BEGIN
   Zulauf_AR_Niv.Bef.BA_Nrm := FALSE;
   Zulauf_AR_Niv.Bef.BA_Frz := FALSE;
   Zulauf_AR_Niv.Bef.BA_EW := FALSE;
   Zulauf_AR_Niv.Bef.BA_Sim := FALSE;
   Zulauf_AR_Niv.Bef.BA_Wart := FALSE;
   Zulauf_AR_Niv.Bef.Frg_HH := FALSE;
   Zulauf_AR_Niv.Bef.Frg_H := FALSE;
   Zulauf_AR_Niv.Bef.Frg_L := FALSE;
   Zulauf_AR_Niv.Bef.Frg_LL := FALSE;
   Zulauf_AR_Niv.Bef.SB_MW_frz := FALSE;
   Zulauf_AR_Niv.Bef.SB_MW_EW := FALSE;
   Zulauf_AR_Niv.Bef.Res_11 := FALSE;
   Zulauf_AR_Niv.Bef.Res_12 := FALSE;
   Zulauf_AR_Niv.Bef.Res_13 := FALSE;
   Zulauf_AR_Niv.Bef.Res_14 := FALSE;
   Zulauf_AR_Niv.Bef.Res_15 := FALSE;
   Zulauf_AR_Niv.Bef.Res_16 := FALSE;
   Zulauf_AR_Niv.Bef.Res_17 := FALSE;
   Zulauf_AR_Niv.Bef.Res_18 := FALSE;
   Zulauf_AR_Niv.Bef.Res_19 := FALSE;
   Zulauf_AR_Niv.Bef.Res_20 := FALSE;
   Zulauf_AR_Niv.Bef.Res_21 := FALSE;
   Zulauf_AR_Niv.Bef.Res_22 := FALSE;
   Zulauf_AR_Niv.Bef.Res_23 := FALSE;
   Zulauf_AR_Niv.Bef.Res_24 := FALSE;
   Zulauf_AR_Niv.Bef.Res_25 := FALSE;
   Zulauf_AR_Niv.Bef.Res_26 := FALSE;
   Zulauf_AR_Niv.Bef.Res_27 := FALSE;
   Zulauf_AR_Niv.Bef.Res_28 := FALSE;
   Zulauf_AR_Niv.Bef.Res_29 := FALSE;
   Zulauf_AR_Niv.Bef.Res_30 := FALSE;
   Zulauf_AR_Niv.Bef.BF_Quit := FALSE;
   Zulauf_AR_Niv.MW_Sim := 8.0;
   Zulauf_AR_Temp.Bef.BA_Nrm := FALSE;
   Zulauf_AR_Temp.Bef.BA_Frz := FALSE;
   Zulauf_AR_Temp.Bef.BA_EW := FALSE;
   Zulauf_AR_Temp.Bef.BA_Sim := FALSE;
   Zulauf_AR_Temp.Bef.BA_Wart := FALSE;
   Zulauf_AR_Temp.Bef.Frg_HH := FALSE;
   Zulauf_AR_Temp.Bef.Frg_H := FALSE;
   Zulauf_AR_Temp.Bef.Frg_L := FALSE;
   Zulauf_AR_Temp.Bef.Frg_LL := FALSE;
   Zulauf_AR_Temp.Bef.SB_MW_frz := FALSE;
   Zulauf_AR_Temp.Bef.SB_MW_EW := FALSE;
   Zulauf_AR_Temp.Bef.Res_11 := FALSE;
   Zulauf_AR_Temp.Bef.Res_12 := FALSE;
   Zulauf_AR_Temp.Bef.Res_13 := FALSE;
   Zulauf_AR_Temp.Bef.Res_14 := FALSE;
   Zulauf_AR_Temp.Bef.Res_15 := FALSE;
   Zulauf_AR_Temp.Bef.Res_16 := FALSE;
   Zulauf_AR_Temp.Bef.Res_17 := FALSE;
   Zulauf_AR_Temp.Bef.Res_18 := FALSE;
   Zulauf_AR_Temp.Bef.Res_19 := FALSE;
   Zulauf_AR_Temp.Bef.Res_20 := FALSE;
   Zulauf_AR_Temp.Bef.Res_21 := FALSE;
   Zulauf_AR_Temp.Bef.Res_22 := FALSE;
   Zulauf_AR_Temp.Bef.Res_23 := FALSE;
   Zulauf_AR_Temp.Bef.Res_24 := FALSE;
   Zulauf_AR_Temp.Bef.Res_25 := FALSE;
   Zulauf_AR_Temp.Bef.Res_26 := FALSE;
   Zulauf_AR_Temp.Bef.Res_27 := FALSE;
   Zulauf_AR_Temp.Bef.Res_28 := FALSE;
   Zulauf_AR_Temp.Bef.Res_29 := FALSE;
   Zulauf_AR_Temp.Bef.Res_30 := FALSE;
   Zulauf_AR_Temp.Bef.BF_Quit := FALSE;
   Zulauf_AR_Temp.MW_Sim := 0.0;
   Zulauf_AR_DF.Bef.BA_Nrm := FALSE;
   Zulauf_AR_DF.Bef.BA_Frz := FALSE;
   Zulauf_AR_DF.Bef.BA_EW := FALSE;
   Zulauf_AR_DF.Bef.BA_Sim := FALSE;
   Zulauf_AR_DF.Bef.BA_Wart := FALSE;
   Zulauf_AR_DF.Bef.Frg_HH := FALSE;
   Zulauf_AR_DF.Bef.Frg_H := FALSE;
   Zulauf_AR_DF.Bef.Frg_L := FALSE;
   Zulauf_AR_DF.Bef.Frg_LL := FALSE;
   Zulauf_AR_DF.Bef.SB_MW_frz := FALSE;
   Zulauf_AR_DF.Bef.SB_MW_EW := FALSE;
   Zulauf_AR_DF.Bef.Res_11 := FALSE;
   Zulauf_AR_DF.Bef.Res_12 := FALSE;
   Zulauf_AR_DF.Bef.Res_13 := FALSE;
   Zulauf_AR_DF.Bef.Res_14 := FALSE;
   Zulauf_AR_DF.Bef.Res_15 := FALSE;
   Zulauf_AR_DF.Bef.Res_16 := FALSE;
   Zulauf_AR_DF.Bef.Res_17 := FALSE;
   Zulauf_AR_DF.Bef.Res_18 := FALSE;
   Zulauf_AR_DF.Bef.Res_19 := FALSE;
   Zulauf_AR_DF.Bef.Res_20 := FALSE;
   Zulauf_AR_DF.Bef.Res_21 := FALSE;
   Zulauf_AR_DF.Bef.Res_22 := FALSE;
   Zulauf_AR_DF.Bef.Res_23 := FALSE;
   Zulauf_AR_DF.Bef.Res_24 := FALSE;
   Zulauf_AR_DF.Bef.Res_25 := FALSE;
   Zulauf_AR_DF.Bef.Res_26 := FALSE;
   Zulauf_AR_DF.Bef.Res_27 := FALSE;
   Zulauf_AR_DF.Bef.Res_28 := FALSE;
   Zulauf_AR_DF.Bef.Res_29 := FALSE;
   Zulauf_AR_DF.Bef.Res_30 := FALSE;
   Zulauf_AR_DF.Bef.BF_Quit := FALSE;
   Zulauf_AR_DF.MW_Sim := 0.0;
   BB1_AS1_SS.Bef.BA_Nrm := FALSE;
   BB1_AS1_SS.Bef.BA_Frz := FALSE;
   BB1_AS1_SS.Bef.BA_EW := FALSE;
   BB1_AS1_SS.Bef.BA_Sim := FALSE;
   BB1_AS1_SS.Bef.BA_Wart := FALSE;
   BB1_AS1_SS.Bef.Frg_HH := FALSE;
   BB1_AS1_SS.Bef.Frg_H := FALSE;
   BB1_AS1_SS.Bef.Frg_L := FALSE;
   BB1_AS1_SS.Bef.Frg_LL := FALSE;
   BB1_AS1_SS.Bef.SB_MW_frz := FALSE;
   BB1_AS1_SS.Bef.SB_MW_EW := FALSE;
   BB1_AS1_SS.Bef.Res_11 := FALSE;
   BB1_AS1_SS.Bef.Res_12 := FALSE;
   BB1_AS1_SS.Bef.Res_13 := FALSE;
   BB1_AS1_SS.Bef.Res_14 := FALSE;
   BB1_AS1_SS.Bef.Res_15 := FALSE;
   BB1_AS1_SS.Bef.Res_16 := FALSE;
   BB1_AS1_SS.Bef.Res_17 := FALSE;
   BB1_AS1_SS.Bef.Res_18 := FALSE;
   BB1_AS1_SS.Bef.Res_19 := FALSE;
   BB1_AS1_SS.Bef.Res_20 := FALSE;
   BB1_AS1_SS.Bef.Res_21 := FALSE;
   BB1_AS1_SS.Bef.Res_22 := FALSE;
   BB1_AS1_SS.Bef.Res_23 := FALSE;
   BB1_AS1_SS.Bef.Res_24 := FALSE;
   BB1_AS1_SS.Bef.Res_25 := FALSE;
   BB1_AS1_SS.Bef.Res_26 := FALSE;
   BB1_AS1_SS.Bef.Res_27 := FALSE;
   BB1_AS1_SS.Bef.Res_28 := FALSE;
   BB1_AS1_SS.Bef.Res_29 := FALSE;
   BB1_AS1_SS.Bef.Res_30 := FALSE;
   BB1_AS1_SS.Bef.BF_Quit := FALSE;
   BB1_AS1_SS.MW_Sim := 0.0;
   BB1_AS2_SS.Bef.BA_Nrm := FALSE;
   BB1_AS2_SS.Bef.BA_Frz := FALSE;
   BB1_AS2_SS.Bef.BA_EW := FALSE;
   BB1_AS2_SS.Bef.BA_Sim := FALSE;
   BB1_AS2_SS.Bef.BA_Wart := FALSE;
   BB1_AS2_SS.Bef.Frg_HH := FALSE;
   BB1_AS2_SS.Bef.Frg_H := FALSE;
   BB1_AS2_SS.Bef.Frg_L := FALSE;
   BB1_AS2_SS.Bef.Frg_LL := FALSE;
   BB1_AS2_SS.Bef.SB_MW_frz := FALSE;
   BB1_AS2_SS.Bef.SB_MW_EW := FALSE;
   BB1_AS2_SS.Bef.Res_11 := FALSE;
   BB1_AS2_SS.Bef.Res_12 := FALSE;
   BB1_AS2_SS.Bef.Res_13 := FALSE;
   BB1_AS2_SS.Bef.Res_14 := FALSE;
   BB1_AS2_SS.Bef.Res_15 := FALSE;
   BB1_AS2_SS.Bef.Res_16 := FALSE;
   BB1_AS2_SS.Bef.Res_17 := FALSE;
   BB1_AS2_SS.Bef.Res_18 := FALSE;
   BB1_AS2_SS.Bef.Res_19 := FALSE;
   BB1_AS2_SS.Bef.Res_20 := FALSE;
   BB1_AS2_SS.Bef.Res_21 := FALSE;
   BB1_AS2_SS.Bef.Res_22 := FALSE;
   BB1_AS2_SS.Bef.Res_23 := FALSE;
   BB1_AS2_SS.Bef.Res_24 := FALSE;
   BB1_AS2_SS.Bef.Res_25 := FALSE;
   BB1_AS2_SS.Bef.Res_26 := FALSE;
   BB1_AS2_SS.Bef.Res_27 := FALSE;
   BB1_AS2_SS.Bef.Res_28 := FALSE;
   BB1_AS2_SS.Bef.Res_29 := FALSE;
   BB1_AS2_SS.Bef.Res_30 := FALSE;
   BB1_AS2_SS.Bef.BF_Quit := FALSE;
   BB1_AS2_SS.MW_Sim := 75.0;
   BB2_AS1_SS.Bef.BA_Nrm := FALSE;
   BB2_AS1_SS.Bef.BA_Frz := FALSE;
   BB2_AS1_SS.Bef.BA_EW := FALSE;
   BB2_AS1_SS.Bef.BA_Sim := FALSE;
   BB2_AS1_SS.Bef.BA_Wart := FALSE;
   BB2_AS1_SS.Bef.Frg_HH := FALSE;
   BB2_AS1_SS.Bef.Frg_H := FALSE;
   BB2_AS1_SS.Bef.Frg_L := FALSE;
   BB2_AS1_SS.Bef.Frg_LL := FALSE;
   BB2_AS1_SS.Bef.SB_MW_frz := FALSE;
   BB2_AS1_SS.Bef.SB_MW_EW := FALSE;
   BB2_AS1_SS.Bef.Res_11 := FALSE;
   BB2_AS1_SS.Bef.Res_12 := FALSE;
   BB2_AS1_SS.Bef.Res_13 := FALSE;
   BB2_AS1_SS.Bef.Res_14 := FALSE;
   BB2_AS1_SS.Bef.Res_15 := FALSE;
   BB2_AS1_SS.Bef.Res_16 := FALSE;
   BB2_AS1_SS.Bef.Res_17 := FALSE;
   BB2_AS1_SS.Bef.Res_18 := FALSE;
   BB2_AS1_SS.Bef.Res_19 := FALSE;
   BB2_AS1_SS.Bef.Res_20 := FALSE;
   BB2_AS1_SS.Bef.Res_21 := FALSE;
   BB2_AS1_SS.Bef.Res_22 := FALSE;
   BB2_AS1_SS.Bef.Res_23 := FALSE;
   BB2_AS1_SS.Bef.Res_24 := FALSE;
   BB2_AS1_SS.Bef.Res_25 := FALSE;
   BB2_AS1_SS.Bef.Res_26 := FALSE;
   BB2_AS1_SS.Bef.Res_27 := FALSE;
   BB2_AS1_SS.Bef.Res_28 := FALSE;
   BB2_AS1_SS.Bef.Res_29 := FALSE;
   BB2_AS1_SS.Bef.Res_30 := FALSE;
   BB2_AS1_SS.Bef.BF_Quit := FALSE;
   BB2_AS1_SS.MW_Sim := 0.0;
   BB2_AS2_SS.Bef.BA_Nrm := FALSE;
   BB2_AS2_SS.Bef.BA_Frz := FALSE;
   BB2_AS2_SS.Bef.BA_EW := FALSE;
   BB2_AS2_SS.Bef.BA_Sim := FALSE;
   BB2_AS2_SS.Bef.BA_Wart := FALSE;
   BB2_AS2_SS.Bef.Frg_HH := FALSE;
   BB2_AS2_SS.Bef.Frg_H := FALSE;
   BB2_AS2_SS.Bef.Frg_L := FALSE;
   BB2_AS2_SS.Bef.Frg_LL := FALSE;
   BB2_AS2_SS.Bef.SB_MW_frz := FALSE;
   BB2_AS2_SS.Bef.SB_MW_EW := FALSE;
   BB2_AS2_SS.Bef.Res_11 := FALSE;
   BB2_AS2_SS.Bef.Res_12 := FALSE;
   BB2_AS2_SS.Bef.Res_13 := FALSE;
   BB2_AS2_SS.Bef.Res_14 := FALSE;
   BB2_AS2_SS.Bef.Res_15 := FALSE;
   BB2_AS2_SS.Bef.Res_16 := FALSE;
   BB2_AS2_SS.Bef.Res_17 := FALSE;
   BB2_AS2_SS.Bef.Res_18 := FALSE;
   BB2_AS2_SS.Bef.Res_19 := FALSE;
   BB2_AS2_SS.Bef.Res_20 := FALSE;
   BB2_AS2_SS.Bef.Res_21 := FALSE;
   BB2_AS2_SS.Bef.Res_22 := FALSE;
   BB2_AS2_SS.Bef.Res_23 := FALSE;
   BB2_AS2_SS.Bef.Res_24 := FALSE;
   BB2_AS2_SS.Bef.Res_25 := FALSE;
   BB2_AS2_SS.Bef.Res_26 := FALSE;
   BB2_AS2_SS.Bef.Res_27 := FALSE;
   BB2_AS2_SS.Bef.Res_28 := FALSE;
   BB2_AS2_SS.Bef.Res_29 := FALSE;
   BB2_AS2_SS.Bef.Res_30 := FALSE;
   BB2_AS2_SS.Bef.BF_Quit := FALSE;
   BB2_AS2_SS.MW_Sim := 0.0;
   BB1_O2.Bef.BA_Nrm := FALSE;
   BB1_O2.Bef.BA_Frz := FALSE;
   BB1_O2.Bef.BA_EW := FALSE;
   BB1_O2.Bef.BA_Sim := FALSE;
   BB1_O2.Bef.BA_Wart := FALSE;
   BB1_O2.Bef.Frg_HH := FALSE;
   BB1_O2.Bef.Frg_H := FALSE;
   BB1_O2.Bef.Frg_L := FALSE;
   BB1_O2.Bef.Frg_LL := FALSE;
   BB1_O2.Bef.SB_MW_frz := FALSE;
   BB1_O2.Bef.SB_MW_EW := FALSE;
   BB1_O2.Bef.Res_11 := FALSE;
   BB1_O2.Bef.Res_12 := FALSE;
   BB1_O2.Bef.Res_13 := FALSE;
   BB1_O2.Bef.Res_14 := FALSE;
   BB1_O2.Bef.Res_15 := FALSE;
   BB1_O2.Bef.Res_16 := FALSE;
   BB1_O2.Bef.Res_17 := FALSE;
   BB1_O2.Bef.Res_18 := FALSE;
   BB1_O2.Bef.Res_19 := FALSE;
   BB1_O2.Bef.Res_20 := FALSE;
   BB1_O2.Bef.Res_21 := FALSE;
   BB1_O2.Bef.Res_22 := FALSE;
   BB1_O2.Bef.Res_23 := FALSE;
   BB1_O2.Bef.Res_24 := FALSE;
   BB1_O2.Bef.Res_25 := FALSE;
   BB1_O2.Bef.Res_26 := FALSE;
   BB1_O2.Bef.Res_27 := FALSE;
   BB1_O2.Bef.Res_28 := FALSE;
   BB1_O2.Bef.Res_29 := FALSE;
   BB1_O2.Bef.Res_30 := FALSE;
   BB1_O2.Bef.BF_Quit := FALSE;
   BB1_O2.MW_Sim := 0.0;
   BB1_Temp.Bef.BA_Nrm := FALSE;
   BB1_Temp.Bef.BA_Frz := FALSE;
   BB1_Temp.Bef.BA_EW := FALSE;
   BB1_Temp.Bef.BA_Sim := FALSE;
   BB1_Temp.Bef.BA_Wart := FALSE;
   BB1_Temp.Bef.Frg_HH := FALSE;
   BB1_Temp.Bef.Frg_H := FALSE;
   BB1_Temp.Bef.Frg_L := FALSE;
   BB1_Temp.Bef.Frg_LL := FALSE;
   BB1_Temp.Bef.SB_MW_frz := FALSE;
   BB1_Temp.Bef.SB_MW_EW := FALSE;
   BB1_Temp.Bef.Res_11 := FALSE;
   BB1_Temp.Bef.Res_12 := FALSE;
   BB1_Temp.Bef.Res_13 := FALSE;
   BB1_Temp.Bef.Res_14 := FALSE;
   BB1_Temp.Bef.Res_15 := FALSE;
   BB1_Temp.Bef.Res_16 := FALSE;
   BB1_Temp.Bef.Res_17 := FALSE;
   BB1_Temp.Bef.Res_18 := FALSE;
   BB1_Temp.Bef.Res_19 := FALSE;
   BB1_Temp.Bef.Res_20 := FALSE;
   BB1_Temp.Bef.Res_21 := FALSE;
   BB1_Temp.Bef.Res_22 := FALSE;
   BB1_Temp.Bef.Res_23 := FALSE;
   BB1_Temp.Bef.Res_24 := FALSE;
   BB1_Temp.Bef.Res_25 := FALSE;
   BB1_Temp.Bef.Res_26 := FALSE;
   BB1_Temp.Bef.Res_27 := FALSE;
   BB1_Temp.Bef.Res_28 := FALSE;
   BB1_Temp.Bef.Res_29 := FALSE;
   BB1_Temp.Bef.Res_30 := FALSE;
   BB1_Temp.Bef.BF_Quit := FALSE;
   BB1_Temp.MW_Sim := 0.0;
   BB2_O2.Bef.BA_Nrm := FALSE;
   BB2_O2.Bef.BA_Frz := FALSE;
   BB2_O2.Bef.BA_EW := FALSE;
   BB2_O2.Bef.BA_Sim := FALSE;
   BB2_O2.Bef.BA_Wart := FALSE;
   BB2_O2.Bef.Frg_HH := FALSE;
   BB2_O2.Bef.Frg_H := FALSE;
   BB2_O2.Bef.Frg_L := FALSE;
   BB2_O2.Bef.Frg_LL := FALSE;
   BB2_O2.Bef.SB_MW_frz := FALSE;
   BB2_O2.Bef.SB_MW_EW := FALSE;
   BB2_O2.Bef.Res_11 := FALSE;
   BB2_O2.Bef.Res_12 := FALSE;
   BB2_O2.Bef.Res_13 := FALSE;
   BB2_O2.Bef.Res_14 := FALSE;
   BB2_O2.Bef.Res_15 := FALSE;
   BB2_O2.Bef.Res_16 := FALSE;
   BB2_O2.Bef.Res_17 := FALSE;
   BB2_O2.Bef.Res_18 := FALSE;
   BB2_O2.Bef.Res_19 := FALSE;
   BB2_O2.Bef.Res_20 := FALSE;
   BB2_O2.Bef.Res_21 := FALSE;
   BB2_O2.Bef.Res_22 := FALSE;
   BB2_O2.Bef.Res_23 := FALSE;
   BB2_O2.Bef.Res_24 := FALSE;
   BB2_O2.Bef.Res_25 := FALSE;
   BB2_O2.Bef.Res_26 := FALSE;
   BB2_O2.Bef.Res_27 := FALSE;
   BB2_O2.Bef.Res_28 := FALSE;
   BB2_O2.Bef.Res_29 := FALSE;
   BB2_O2.Bef.Res_30 := FALSE;
   BB2_O2.Bef.BF_Quit := FALSE;
   BB2_O2.MW_Sim := 0.0;
   BB2_Temp.Bef.BA_Nrm := FALSE;
   BB2_Temp.Bef.BA_Frz := FALSE;
   BB2_Temp.Bef.BA_EW := FALSE;
   BB2_Temp.Bef.BA_Sim := FALSE;
   BB2_Temp.Bef.BA_Wart := FALSE;
   BB2_Temp.Bef.Frg_HH := FALSE;
   BB2_Temp.Bef.Frg_H := FALSE;
   BB2_Temp.Bef.Frg_L := FALSE;
   BB2_Temp.Bef.Frg_LL := FALSE;
   BB2_Temp.Bef.SB_MW_frz := FALSE;
   BB2_Temp.Bef.SB_MW_EW := FALSE;
   BB2_Temp.Bef.Res_11 := FALSE;
   BB2_Temp.Bef.Res_12 := FALSE;
   BB2_Temp.Bef.Res_13 := FALSE;
   BB2_Temp.Bef.Res_14 := FALSE;
   BB2_Temp.Bef.Res_15 := FALSE;
   BB2_Temp.Bef.Res_16 := FALSE;
   BB2_Temp.Bef.Res_17 := FALSE;
   BB2_Temp.Bef.Res_18 := FALSE;
   BB2_Temp.Bef.Res_19 := FALSE;
   BB2_Temp.Bef.Res_20 := FALSE;
   BB2_Temp.Bef.Res_21 := FALSE;
   BB2_Temp.Bef.Res_22 := FALSE;
   BB2_Temp.Bef.Res_23 := FALSE;
   BB2_Temp.Bef.Res_24 := FALSE;
   BB2_Temp.Bef.Res_25 := FALSE;
   BB2_Temp.Bef.Res_26 := FALSE;
   BB2_Temp.Bef.Res_27 := FALSE;
   BB2_Temp.Bef.Res_28 := FALSE;
   BB2_Temp.Bef.Res_29 := FALSE;
   BB2_Temp.Bef.Res_30 := FALSE;
   BB2_Temp.Bef.BF_Quit := FALSE;
   BB2_Temp.MW_Sim := 0.0;
   BB1_DF.Bef.BA_Nrm := FALSE;
   BB1_DF.Bef.BA_Frz := FALSE;
   BB1_DF.Bef.BA_EW := FALSE;
   BB1_DF.Bef.BA_Sim := FALSE;
   BB1_DF.Bef.BA_Wart := FALSE;
   BB1_DF.Bef.Frg_HH := FALSE;
   BB1_DF.Bef.Frg_H := FALSE;
   BB1_DF.Bef.Frg_L := FALSE;
   BB1_DF.Bef.Frg_LL := FALSE;
   BB1_DF.Bef.SB_MW_frz := FALSE;
   BB1_DF.Bef.SB_MW_EW := FALSE;
   BB1_DF.Bef.Res_11 := FALSE;
   BB1_DF.Bef.Res_12 := FALSE;
   BB1_DF.Bef.Res_13 := FALSE;
   BB1_DF.Bef.Res_14 := FALSE;
   BB1_DF.Bef.Res_15 := FALSE;
   BB1_DF.Bef.Res_16 := FALSE;
   BB1_DF.Bef.Res_17 := FALSE;
   BB1_DF.Bef.Res_18 := FALSE;
   BB1_DF.Bef.Res_19 := FALSE;
   BB1_DF.Bef.Res_20 := FALSE;
   BB1_DF.Bef.Res_21 := FALSE;
   BB1_DF.Bef.Res_22 := FALSE;
   BB1_DF.Bef.Res_23 := FALSE;
   BB1_DF.Bef.Res_24 := FALSE;
   BB1_DF.Bef.Res_25 := FALSE;
   BB1_DF.Bef.Res_26 := FALSE;
   BB1_DF.Bef.Res_27 := FALSE;
   BB1_DF.Bef.Res_28 := FALSE;
   BB1_DF.Bef.Res_29 := FALSE;
   BB1_DF.Bef.Res_30 := FALSE;
   BB1_DF.Bef.BF_Quit := FALSE;
   BB1_DF.MW_Sim := 0.0;
   BB2_DF.Bef.BA_Nrm := FALSE;
   BB2_DF.Bef.BA_Frz := FALSE;
   BB2_DF.Bef.BA_EW := FALSE;
   BB2_DF.Bef.BA_Sim := FALSE;
   BB2_DF.Bef.BA_Wart := FALSE;
   BB2_DF.Bef.Frg_HH := FALSE;
   BB2_DF.Bef.Frg_H := FALSE;
   BB2_DF.Bef.Frg_L := FALSE;
   BB2_DF.Bef.Frg_LL := FALSE;
   BB2_DF.Bef.SB_MW_frz := FALSE;
   BB2_DF.Bef.SB_MW_EW := FALSE;
   BB2_DF.Bef.Res_11 := FALSE;
   BB2_DF.Bef.Res_12 := FALSE;
   BB2_DF.Bef.Res_13 := FALSE;
   BB2_DF.Bef.Res_14 := FALSE;
   BB2_DF.Bef.Res_15 := FALSE;
   BB2_DF.Bef.Res_16 := FALSE;
   BB2_DF.Bef.Res_17 := FALSE;
   BB2_DF.Bef.Res_18 := FALSE;
   BB2_DF.Bef.Res_19 := FALSE;
   BB2_DF.Bef.Res_20 := FALSE;
   BB2_DF.Bef.Res_21 := FALSE;
   BB2_DF.Bef.Res_22 := FALSE;
   BB2_DF.Bef.Res_23 := FALSE;
   BB2_DF.Bef.Res_24 := FALSE;
   BB2_DF.Bef.Res_25 := FALSE;
   BB2_DF.Bef.Res_26 := FALSE;
   BB2_DF.Bef.Res_27 := FALSE;
   BB2_DF.Bef.Res_28 := FALSE;
   BB2_DF.Bef.Res_29 := FALSE;
   BB2_DF.Bef.Res_30 := FALSE;
   BB2_DF.Bef.BF_Quit := FALSE;
   BB2_DF.MW_Sim := 0.0;
   Zulauf_Niv.Bef.BA_Nrm := FALSE;
   Zulauf_Niv.Bef.BA_Frz := FALSE;
   Zulauf_Niv.Bef.BA_EW := FALSE;
   Zulauf_Niv.Bef.BA_Sim := FALSE;
   Zulauf_Niv.Bef.BA_Wart := FALSE;
   Zulauf_Niv.Bef.Frg_HH := FALSE;
   Zulauf_Niv.Bef.Frg_H := FALSE;
   Zulauf_Niv.Bef.Frg_L := FALSE;
   Zulauf_Niv.Bef.Frg_LL := FALSE;
   Zulauf_Niv.Bef.SB_MW_frz := FALSE;
   Zulauf_Niv.Bef.SB_MW_EW := FALSE;
   Zulauf_Niv.Bef.Res_11 := FALSE;
   Zulauf_Niv.Bef.Res_12 := FALSE;
   Zulauf_Niv.Bef.Res_13 := FALSE;
   Zulauf_Niv.Bef.Res_14 := FALSE;
   Zulauf_Niv.Bef.Res_15 := FALSE;
   Zulauf_Niv.Bef.Res_16 := FALSE;
   Zulauf_Niv.Bef.Res_17 := FALSE;
   Zulauf_Niv.Bef.Res_18 := FALSE;
   Zulauf_Niv.Bef.Res_19 := FALSE;
   Zulauf_Niv.Bef.Res_20 := FALSE;
   Zulauf_Niv.Bef.Res_21 := FALSE;
   Zulauf_Niv.Bef.Res_22 := FALSE;
   Zulauf_Niv.Bef.Res_23 := FALSE;
   Zulauf_Niv.Bef.Res_24 := FALSE;
   Zulauf_Niv.Bef.Res_25 := FALSE;
   Zulauf_Niv.Bef.Res_26 := FALSE;
   Zulauf_Niv.Bef.Res_27 := FALSE;
   Zulauf_Niv.Bef.Res_28 := FALSE;
   Zulauf_Niv.Bef.Res_29 := FALSE;
   Zulauf_Niv.Bef.Res_30 := FALSE;
   Zulauf_Niv.Bef.BF_Quit := FALSE;
   Zulauf_Niv.MW_Sim := 0.6;
   Zulauf_DF.Bef.BA_Nrm := FALSE;
   Zulauf_DF.Bef.BA_Frz := FALSE;
   Zulauf_DF.Bef.BA_EW := FALSE;
   Zulauf_DF.Bef.BA_Sim := FALSE;
   Zulauf_DF.Bef.BA_Wart := FALSE;
   Zulauf_DF.Bef.Frg_HH := FALSE;
   Zulauf_DF.Bef.Frg_H := FALSE;
   Zulauf_DF.Bef.Frg_L := FALSE;
   Zulauf_DF.Bef.Frg_LL := FALSE;
   Zulauf_DF.Bef.SB_MW_frz := FALSE;
   Zulauf_DF.Bef.SB_MW_EW := FALSE;
   Zulauf_DF.Bef.Res_11 := FALSE;
   Zulauf_DF.Bef.Res_12 := FALSE;
   Zulauf_DF.Bef.Res_13 := FALSE;
   Zulauf_DF.Bef.Res_14 := FALSE;
   Zulauf_DF.Bef.Res_15 := FALSE;
   Zulauf_DF.Bef.Res_16 := FALSE;
   Zulauf_DF.Bef.Res_17 := FALSE;
   Zulauf_DF.Bef.Res_18 := FALSE;
   Zulauf_DF.Bef.Res_19 := FALSE;
   Zulauf_DF.Bef.Res_20 := FALSE;
   Zulauf_DF.Bef.Res_21 := FALSE;
   Zulauf_DF.Bef.Res_22 := FALSE;
   Zulauf_DF.Bef.Res_23 := FALSE;
   Zulauf_DF.Bef.Res_24 := FALSE;
   Zulauf_DF.Bef.Res_25 := FALSE;
   Zulauf_DF.Bef.Res_26 := FALSE;
   Zulauf_DF.Bef.Res_27 := FALSE;
   Zulauf_DF.Bef.Res_28 := FALSE;
   Zulauf_DF.Bef.Res_29 := FALSE;
   Zulauf_DF.Bef.Res_30 := FALSE;
   Zulauf_DF.Bef.BF_Quit := FALSE;
   Zulauf_DF.MW_Sim := 0.0;
   Verteiler_pH.Bef.BA_Nrm := FALSE;
   Verteiler_pH.Bef.BA_Frz := FALSE;
   Verteiler_pH.Bef.BA_EW := FALSE;
   Verteiler_pH.Bef.BA_Sim := FALSE;
   Verteiler_pH.Bef.BA_Wart := FALSE;
   Verteiler_pH.Bef.Frg_HH := FALSE;
   Verteiler_pH.Bef.Frg_H := FALSE;
   Verteiler_pH.Bef.Frg_L := FALSE;
   Verteiler_pH.Bef.Frg_LL := FALSE;
   Verteiler_pH.Bef.SB_MW_frz := FALSE;
   Verteiler_pH.Bef.SB_MW_EW := FALSE;
   Verteiler_pH.Bef.Res_11 := FALSE;
   Verteiler_pH.Bef.Res_12 := FALSE;
   Verteiler_pH.Bef.Res_13 := FALSE;
   Verteiler_pH.Bef.Res_14 := FALSE;
   Verteiler_pH.Bef.Res_15 := FALSE;
   Verteiler_pH.Bef.Res_16 := FALSE;
   Verteiler_pH.Bef.Res_17 := FALSE;
   Verteiler_pH.Bef.Res_18 := FALSE;
   Verteiler_pH.Bef.Res_19 := FALSE;
   Verteiler_pH.Bef.Res_20 := FALSE;
   Verteiler_pH.Bef.Res_21 := FALSE;
   Verteiler_pH.Bef.Res_22 := FALSE;
   Verteiler_pH.Bef.Res_23 := FALSE;
   Verteiler_pH.Bef.Res_24 := FALSE;
   Verteiler_pH.Bef.Res_25 := FALSE;
   Verteiler_pH.Bef.Res_26 := FALSE;
   Verteiler_pH.Bef.Res_27 := FALSE;
   Verteiler_pH.Bef.Res_28 := FALSE;
   Verteiler_pH.Bef.Res_29 := FALSE;
   Verteiler_pH.Bef.Res_30 := FALSE;
   Verteiler_pH.Bef.BF_Quit := FALSE;
   Verteiler_pH.MW_Sim := 7.6;
   Verteiler_O2.Bef.BA_Nrm := FALSE;
   Verteiler_O2.Bef.BA_Frz := FALSE;
   Verteiler_O2.Bef.BA_EW := FALSE;
   Verteiler_O2.Bef.BA_Sim := FALSE;
   Verteiler_O2.Bef.BA_Wart := FALSE;
   Verteiler_O2.Bef.Frg_HH := FALSE;
   Verteiler_O2.Bef.Frg_H := FALSE;
   Verteiler_O2.Bef.Frg_L := FALSE;
   Verteiler_O2.Bef.Frg_LL := FALSE;
   Verteiler_O2.Bef.SB_MW_frz := FALSE;
   Verteiler_O2.Bef.SB_MW_EW := FALSE;
   Verteiler_O2.Bef.Res_11 := FALSE;
   Verteiler_O2.Bef.Res_12 := FALSE;
   Verteiler_O2.Bef.Res_13 := FALSE;
   Verteiler_O2.Bef.Res_14 := FALSE;
   Verteiler_O2.Bef.Res_15 := FALSE;
   Verteiler_O2.Bef.Res_16 := FALSE;
   Verteiler_O2.Bef.Res_17 := FALSE;
   Verteiler_O2.Bef.Res_18 := FALSE;
   Verteiler_O2.Bef.Res_19 := FALSE;
   Verteiler_O2.Bef.Res_20 := FALSE;
   Verteiler_O2.Bef.Res_21 := FALSE;
   Verteiler_O2.Bef.Res_22 := FALSE;
   Verteiler_O2.Bef.Res_23 := FALSE;
   Verteiler_O2.Bef.Res_24 := FALSE;
   Verteiler_O2.Bef.Res_25 := FALSE;
   Verteiler_O2.Bef.Res_26 := FALSE;
   Verteiler_O2.Bef.Res_27 := FALSE;
   Verteiler_O2.Bef.Res_28 := FALSE;
   Verteiler_O2.Bef.Res_29 := FALSE;
   Verteiler_O2.Bef.Res_30 := FALSE;
   Verteiler_O2.Bef.BF_Quit := FALSE;
   Verteiler_O2.MW_Sim := 5.8;
   Verteiler_Temp.Bef.BA_Nrm := FALSE;
   Verteiler_Temp.Bef.BA_Frz := FALSE;
   Verteiler_Temp.Bef.BA_EW := FALSE;
   Verteiler_Temp.Bef.BA_Sim := FALSE;
   Verteiler_Temp.Bef.BA_Wart := FALSE;
   Verteiler_Temp.Bef.Frg_HH := FALSE;
   Verteiler_Temp.Bef.Frg_H := FALSE;
   Verteiler_Temp.Bef.Frg_L := FALSE;
   Verteiler_Temp.Bef.Frg_LL := FALSE;
   Verteiler_Temp.Bef.SB_MW_frz := FALSE;
   Verteiler_Temp.Bef.SB_MW_EW := FALSE;
   Verteiler_Temp.Bef.Res_11 := FALSE;
   Verteiler_Temp.Bef.Res_12 := FALSE;
   Verteiler_Temp.Bef.Res_13 := FALSE;
   Verteiler_Temp.Bef.Res_14 := FALSE;
   Verteiler_Temp.Bef.Res_15 := FALSE;
   Verteiler_Temp.Bef.Res_16 := FALSE;
   Verteiler_Temp.Bef.Res_17 := FALSE;
   Verteiler_Temp.Bef.Res_18 := FALSE;
   Verteiler_Temp.Bef.Res_19 := FALSE;
   Verteiler_Temp.Bef.Res_20 := FALSE;
   Verteiler_Temp.Bef.Res_21 := FALSE;
   Verteiler_Temp.Bef.Res_22 := FALSE;
   Verteiler_Temp.Bef.Res_23 := FALSE;
   Verteiler_Temp.Bef.Res_24 := FALSE;
   Verteiler_Temp.Bef.Res_25 := FALSE;
   Verteiler_Temp.Bef.Res_26 := FALSE;
   Verteiler_Temp.Bef.Res_27 := FALSE;
   Verteiler_Temp.Bef.Res_28 := FALSE;
   Verteiler_Temp.Bef.Res_29 := FALSE;
   Verteiler_Temp.Bef.Res_30 := FALSE;
   Verteiler_Temp.Bef.BF_Quit := FALSE;
   Verteiler_Temp.MW_Sim := 21.0;
   BB_UeSS_DF.Bef.BA_Nrm := FALSE;
   BB_UeSS_DF.Bef.BA_Frz := FALSE;
   BB_UeSS_DF.Bef.BA_EW := FALSE;
   BB_UeSS_DF.Bef.BA_Sim := FALSE;
   BB_UeSS_DF.Bef.BA_Wart := FALSE;
   BB_UeSS_DF.Bef.Frg_HH := FALSE;
   BB_UeSS_DF.Bef.Frg_H := FALSE;
   BB_UeSS_DF.Bef.Frg_L := FALSE;
   BB_UeSS_DF.Bef.Frg_LL := FALSE;
   BB_UeSS_DF.Bef.SB_MW_frz := FALSE;
   BB_UeSS_DF.Bef.SB_MW_EW := FALSE;
   BB_UeSS_DF.Bef.Res_11 := FALSE;
   BB_UeSS_DF.Bef.Res_12 := FALSE;
   BB_UeSS_DF.Bef.Res_13 := FALSE;
   BB_UeSS_DF.Bef.Res_14 := FALSE;
   BB_UeSS_DF.Bef.Res_15 := FALSE;
   BB_UeSS_DF.Bef.Res_16 := FALSE;
   BB_UeSS_DF.Bef.Res_17 := FALSE;
   BB_UeSS_DF.Bef.Res_18 := FALSE;
   BB_UeSS_DF.Bef.Res_19 := FALSE;
   BB_UeSS_DF.Bef.Res_20 := FALSE;
   BB_UeSS_DF.Bef.Res_21 := FALSE;
   BB_UeSS_DF.Bef.Res_22 := FALSE;
   BB_UeSS_DF.Bef.Res_23 := FALSE;
   BB_UeSS_DF.Bef.Res_24 := FALSE;
   BB_UeSS_DF.Bef.Res_25 := FALSE;
   BB_UeSS_DF.Bef.Res_26 := FALSE;
   BB_UeSS_DF.Bef.Res_27 := FALSE;
   BB_UeSS_DF.Bef.Res_28 := FALSE;
   BB_UeSS_DF.Bef.Res_29 := FALSE;
   BB_UeSS_DF.Bef.Res_30 := FALSE;
   BB_UeSS_DF.Bef.BF_Quit := FALSE;
   BB_UeSS_DF.MW_Sim := 0.0;
   Ablauf_DF.Bef.BA_Nrm := FALSE;
   Ablauf_DF.Bef.BA_Frz := FALSE;
   Ablauf_DF.Bef.BA_EW := FALSE;
   Ablauf_DF.Bef.BA_Sim := FALSE;
   Ablauf_DF.Bef.BA_Wart := FALSE;
   Ablauf_DF.Bef.Frg_HH := FALSE;
   Ablauf_DF.Bef.Frg_H := FALSE;
   Ablauf_DF.Bef.Frg_L := FALSE;
   Ablauf_DF.Bef.Frg_LL := FALSE;
   Ablauf_DF.Bef.SB_MW_frz := FALSE;
   Ablauf_DF.Bef.SB_MW_EW := FALSE;
   Ablauf_DF.Bef.Res_11 := FALSE;
   Ablauf_DF.Bef.Res_12 := FALSE;
   Ablauf_DF.Bef.Res_13 := FALSE;
   Ablauf_DF.Bef.Res_14 := FALSE;
   Ablauf_DF.Bef.Res_15 := FALSE;
   Ablauf_DF.Bef.Res_16 := FALSE;
   Ablauf_DF.Bef.Res_17 := FALSE;
   Ablauf_DF.Bef.Res_18 := FALSE;
   Ablauf_DF.Bef.Res_19 := FALSE;
   Ablauf_DF.Bef.Res_20 := FALSE;
   Ablauf_DF.Bef.Res_21 := FALSE;
   Ablauf_DF.Bef.Res_22 := FALSE;
   Ablauf_DF.Bef.Res_23 := FALSE;
   Ablauf_DF.Bef.Res_24 := FALSE;
   Ablauf_DF.Bef.Res_25 := FALSE;
   Ablauf_DF.Bef.Res_26 := FALSE;
   Ablauf_DF.Bef.Res_27 := FALSE;
   Ablauf_DF.Bef.Res_28 := FALSE;
   Ablauf_DF.Bef.Res_29 := FALSE;
   Ablauf_DF.Bef.Res_30 := FALSE;
   Ablauf_DF.Bef.BF_Quit := FALSE;
   Ablauf_DF.MW_Sim := 0.0;
   Ablauf_pH.Bef.BA_Nrm := FALSE;
   Ablauf_pH.Bef.BA_Frz := FALSE;
   Ablauf_pH.Bef.BA_EW := FALSE;
   Ablauf_pH.Bef.BA_Sim := FALSE;
   Ablauf_pH.Bef.BA_Wart := FALSE;
   Ablauf_pH.Bef.Frg_HH := FALSE;
   Ablauf_pH.Bef.Frg_H := FALSE;
   Ablauf_pH.Bef.Frg_L := FALSE;
   Ablauf_pH.Bef.Frg_LL := FALSE;
   Ablauf_pH.Bef.SB_MW_frz := FALSE;
   Ablauf_pH.Bef.SB_MW_EW := FALSE;
   Ablauf_pH.Bef.Res_11 := FALSE;
   Ablauf_pH.Bef.Res_12 := FALSE;
   Ablauf_pH.Bef.Res_13 := FALSE;
   Ablauf_pH.Bef.Res_14 := FALSE;
   Ablauf_pH.Bef.Res_15 := FALSE;
   Ablauf_pH.Bef.Res_16 := FALSE;
   Ablauf_pH.Bef.Res_17 := FALSE;
   Ablauf_pH.Bef.Res_18 := FALSE;
   Ablauf_pH.Bef.Res_19 := FALSE;
   Ablauf_pH.Bef.Res_20 := FALSE;
   Ablauf_pH.Bef.Res_21 := FALSE;
   Ablauf_pH.Bef.Res_22 := FALSE;
   Ablauf_pH.Bef.Res_23 := FALSE;
   Ablauf_pH.Bef.Res_24 := FALSE;
   Ablauf_pH.Bef.Res_25 := FALSE;
   Ablauf_pH.Bef.Res_26 := FALSE;
   Ablauf_pH.Bef.Res_27 := FALSE;
   Ablauf_pH.Bef.Res_28 := FALSE;
   Ablauf_pH.Bef.Res_29 := FALSE;
   Ablauf_pH.Bef.Res_30 := FALSE;
   Ablauf_pH.Bef.BF_Quit := FALSE;
   Ablauf_pH.MW_Sim := 0.0;
   Ablauf_O2.Bef.BA_Nrm := FALSE;
   Ablauf_O2.Bef.BA_Frz := FALSE;
   Ablauf_O2.Bef.BA_EW := FALSE;
   Ablauf_O2.Bef.BA_Sim := FALSE;
   Ablauf_O2.Bef.BA_Wart := FALSE;
   Ablauf_O2.Bef.Frg_HH := FALSE;
   Ablauf_O2.Bef.Frg_H := FALSE;
   Ablauf_O2.Bef.Frg_L := FALSE;
   Ablauf_O2.Bef.Frg_LL := FALSE;
   Ablauf_O2.Bef.SB_MW_frz := FALSE;
   Ablauf_O2.Bef.SB_MW_EW := FALSE;
   Ablauf_O2.Bef.Res_11 := FALSE;
   Ablauf_O2.Bef.Res_12 := FALSE;
   Ablauf_O2.Bef.Res_13 := FALSE;
   Ablauf_O2.Bef.Res_14 := FALSE;
   Ablauf_O2.Bef.Res_15 := FALSE;
   Ablauf_O2.Bef.Res_16 := FALSE;
   Ablauf_O2.Bef.Res_17 := FALSE;
   Ablauf_O2.Bef.Res_18 := FALSE;
   Ablauf_O2.Bef.Res_19 := FALSE;
   Ablauf_O2.Bef.Res_20 := FALSE;
   Ablauf_O2.Bef.Res_21 := FALSE;
   Ablauf_O2.Bef.Res_22 := FALSE;
   Ablauf_O2.Bef.Res_23 := FALSE;
   Ablauf_O2.Bef.Res_24 := FALSE;
   Ablauf_O2.Bef.Res_25 := FALSE;
   Ablauf_O2.Bef.Res_26 := FALSE;
   Ablauf_O2.Bef.Res_27 := FALSE;
   Ablauf_O2.Bef.Res_28 := FALSE;
   Ablauf_O2.Bef.Res_29 := FALSE;
   Ablauf_O2.Bef.Res_30 := FALSE;
   Ablauf_O2.Bef.BF_Quit := FALSE;
   Ablauf_O2.MW_Sim := 0.0;
   Ablauf_Temp.Bef.BA_Nrm := FALSE;
   Ablauf_Temp.Bef.BA_Frz := FALSE;
   Ablauf_Temp.Bef.BA_EW := FALSE;
   Ablauf_Temp.Bef.BA_Sim := FALSE;
   Ablauf_Temp.Bef.BA_Wart := FALSE;
   Ablauf_Temp.Bef.Frg_HH := FALSE;
   Ablauf_Temp.Bef.Frg_H := FALSE;
   Ablauf_Temp.Bef.Frg_L := FALSE;
   Ablauf_Temp.Bef.Frg_LL := FALSE;
   Ablauf_Temp.Bef.SB_MW_frz := FALSE;
   Ablauf_Temp.Bef.SB_MW_EW := FALSE;
   Ablauf_Temp.Bef.Res_11 := FALSE;
   Ablauf_Temp.Bef.Res_12 := FALSE;
   Ablauf_Temp.Bef.Res_13 := FALSE;
   Ablauf_Temp.Bef.Res_14 := FALSE;
   Ablauf_Temp.Bef.Res_15 := FALSE;
   Ablauf_Temp.Bef.Res_16 := FALSE;
   Ablauf_Temp.Bef.Res_17 := FALSE;
   Ablauf_Temp.Bef.Res_18 := FALSE;
   Ablauf_Temp.Bef.Res_19 := FALSE;
   Ablauf_Temp.Bef.Res_20 := FALSE;
   Ablauf_Temp.Bef.Res_21 := FALSE;
   Ablauf_Temp.Bef.Res_22 := FALSE;
   Ablauf_Temp.Bef.Res_23 := FALSE;
   Ablauf_Temp.Bef.Res_24 := FALSE;
   Ablauf_Temp.Bef.Res_25 := FALSE;
   Ablauf_Temp.Bef.Res_26 := FALSE;
   Ablauf_Temp.Bef.Res_27 := FALSE;
   Ablauf_Temp.Bef.Res_28 := FALSE;
   Ablauf_Temp.Bef.Res_29 := FALSE;
   Ablauf_Temp.Bef.Res_30 := FALSE;
   Ablauf_Temp.Bef.BF_Quit := FALSE;
   Ablauf_Temp.MW_Sim := 0.0;
   Schlamm_ED_Niv.Bef.BA_Nrm := FALSE;
   Schlamm_ED_Niv.Bef.BA_Frz := FALSE;
   Schlamm_ED_Niv.Bef.BA_EW := FALSE;
   Schlamm_ED_Niv.Bef.BA_Sim := FALSE;
   Schlamm_ED_Niv.Bef.BA_Wart := FALSE;
   Schlamm_ED_Niv.Bef.Frg_HH := FALSE;
   Schlamm_ED_Niv.Bef.Frg_H := FALSE;
   Schlamm_ED_Niv.Bef.Frg_L := FALSE;
   Schlamm_ED_Niv.Bef.Frg_LL := FALSE;
   Schlamm_ED_Niv.Bef.SB_MW_frz := FALSE;
   Schlamm_ED_Niv.Bef.SB_MW_EW := FALSE;
   Schlamm_ED_Niv.Bef.Res_11 := FALSE;
   Schlamm_ED_Niv.Bef.Res_12 := FALSE;
   Schlamm_ED_Niv.Bef.Res_13 := FALSE;
   Schlamm_ED_Niv.Bef.Res_14 := FALSE;
   Schlamm_ED_Niv.Bef.Res_15 := FALSE;
   Schlamm_ED_Niv.Bef.Res_16 := FALSE;
   Schlamm_ED_Niv.Bef.Res_17 := FALSE;
   Schlamm_ED_Niv.Bef.Res_18 := FALSE;
   Schlamm_ED_Niv.Bef.Res_19 := FALSE;
   Schlamm_ED_Niv.Bef.Res_20 := FALSE;
   Schlamm_ED_Niv.Bef.Res_21 := FALSE;
   Schlamm_ED_Niv.Bef.Res_22 := FALSE;
   Schlamm_ED_Niv.Bef.Res_23 := FALSE;
   Schlamm_ED_Niv.Bef.Res_24 := FALSE;
   Schlamm_ED_Niv.Bef.Res_25 := FALSE;
   Schlamm_ED_Niv.Bef.Res_26 := FALSE;
   Schlamm_ED_Niv.Bef.Res_27 := FALSE;
   Schlamm_ED_Niv.Bef.Res_28 := FALSE;
   Schlamm_ED_Niv.Bef.Res_29 := FALSE;
   Schlamm_ED_Niv.Bef.Res_30 := FALSE;
   Schlamm_ED_Niv.Bef.BF_Quit := FALSE;
   Schlamm_ED_Niv.MW_Sim := 0.0;
   Schlamm_Besch_Niv.Bef.BA_Nrm := FALSE;
   Schlamm_Besch_Niv.Bef.BA_Frz := FALSE;
   Schlamm_Besch_Niv.Bef.BA_EW := FALSE;
   Schlamm_Besch_Niv.Bef.BA_Sim := FALSE;
   Schlamm_Besch_Niv.Bef.BA_Wart := FALSE;
   Schlamm_Besch_Niv.Bef.Frg_HH := FALSE;
   Schlamm_Besch_Niv.Bef.Frg_H := FALSE;
   Schlamm_Besch_Niv.Bef.Frg_L := FALSE;
   Schlamm_Besch_Niv.Bef.Frg_LL := FALSE;
   Schlamm_Besch_Niv.Bef.SB_MW_frz := FALSE;
   Schlamm_Besch_Niv.Bef.SB_MW_EW := FALSE;
   Schlamm_Besch_Niv.Bef.Res_11 := FALSE;
   Schlamm_Besch_Niv.Bef.Res_12 := FALSE;
   Schlamm_Besch_Niv.Bef.Res_13 := FALSE;
   Schlamm_Besch_Niv.Bef.Res_14 := FALSE;
   Schlamm_Besch_Niv.Bef.Res_15 := FALSE;
   Schlamm_Besch_Niv.Bef.Res_16 := FALSE;
   Schlamm_Besch_Niv.Bef.Res_17 := FALSE;
   Schlamm_Besch_Niv.Bef.Res_18 := FALSE;
   Schlamm_Besch_Niv.Bef.Res_19 := FALSE;
   Schlamm_Besch_Niv.Bef.Res_20 := FALSE;
   Schlamm_Besch_Niv.Bef.Res_21 := FALSE;
   Schlamm_Besch_Niv.Bef.Res_22 := FALSE;
   Schlamm_Besch_Niv.Bef.Res_23 := FALSE;
   Schlamm_Besch_Niv.Bef.Res_24 := FALSE;
   Schlamm_Besch_Niv.Bef.Res_25 := FALSE;
   Schlamm_Besch_Niv.Bef.Res_26 := FALSE;
   Schlamm_Besch_Niv.Bef.Res_27 := FALSE;
   Schlamm_Besch_Niv.Bef.Res_28 := FALSE;
   Schlamm_Besch_Niv.Bef.Res_29 := FALSE;
   Schlamm_Besch_Niv.Bef.Res_30 := FALSE;
   Schlamm_Besch_Niv.Bef.BF_Quit := FALSE;
   Schlamm_Besch_Niv.MW_Sim := 0.0;
   Schlamm_Besch_DF.Bef.BA_Nrm := FALSE;
   Schlamm_Besch_DF.Bef.BA_Frz := FALSE;
   Schlamm_Besch_DF.Bef.BA_EW := FALSE;
   Schlamm_Besch_DF.Bef.BA_Sim := FALSE;
   Schlamm_Besch_DF.Bef.BA_Wart := FALSE;
   Schlamm_Besch_DF.Bef.Frg_HH := FALSE;
   Schlamm_Besch_DF.Bef.Frg_H := FALSE;
   Schlamm_Besch_DF.Bef.Frg_L := FALSE;
   Schlamm_Besch_DF.Bef.Frg_LL := FALSE;
   Schlamm_Besch_DF.Bef.SB_MW_frz := FALSE;
   Schlamm_Besch_DF.Bef.SB_MW_EW := FALSE;
   Schlamm_Besch_DF.Bef.Res_11 := FALSE;
   Schlamm_Besch_DF.Bef.Res_12 := FALSE;
   Schlamm_Besch_DF.Bef.Res_13 := FALSE;
   Schlamm_Besch_DF.Bef.Res_14 := FALSE;
   Schlamm_Besch_DF.Bef.Res_15 := FALSE;
   Schlamm_Besch_DF.Bef.Res_16 := FALSE;
   Schlamm_Besch_DF.Bef.Res_17 := FALSE;
   Schlamm_Besch_DF.Bef.Res_18 := FALSE;
   Schlamm_Besch_DF.Bef.Res_19 := FALSE;
   Schlamm_Besch_DF.Bef.Res_20 := FALSE;
   Schlamm_Besch_DF.Bef.Res_21 := FALSE;
   Schlamm_Besch_DF.Bef.Res_22 := FALSE;
   Schlamm_Besch_DF.Bef.Res_23 := FALSE;
   Schlamm_Besch_DF.Bef.Res_24 := FALSE;
   Schlamm_Besch_DF.Bef.Res_25 := FALSE;
   Schlamm_Besch_DF.Bef.Res_26 := FALSE;
   Schlamm_Besch_DF.Bef.Res_27 := FALSE;
   Schlamm_Besch_DF.Bef.Res_28 := FALSE;
   Schlamm_Besch_DF.Bef.Res_29 := FALSE;
   Schlamm_Besch_DF.Bef.Res_30 := FALSE;
   Schlamm_Besch_DF.Bef.BF_Quit := FALSE;
   Schlamm_Besch_DF.MW_Sim := 0.0;
   Truebwasser_Niv.Bef.BA_Nrm := FALSE;
   Truebwasser_Niv.Bef.BA_Frz := FALSE;
   Truebwasser_Niv.Bef.BA_EW := FALSE;
   Truebwasser_Niv.Bef.BA_Sim := FALSE;
   Truebwasser_Niv.Bef.BA_Wart := FALSE;
   Truebwasser_Niv.Bef.Frg_HH := FALSE;
   Truebwasser_Niv.Bef.Frg_H := FALSE;
   Truebwasser_Niv.Bef.Frg_L := FALSE;
   Truebwasser_Niv.Bef.Frg_LL := FALSE;
   Truebwasser_Niv.Bef.SB_MW_frz := FALSE;
   Truebwasser_Niv.Bef.SB_MW_EW := FALSE;
   Truebwasser_Niv.Bef.Res_11 := FALSE;
   Truebwasser_Niv.Bef.Res_12 := FALSE;
   Truebwasser_Niv.Bef.Res_13 := FALSE;
   Truebwasser_Niv.Bef.Res_14 := FALSE;
   Truebwasser_Niv.Bef.Res_15 := FALSE;
   Truebwasser_Niv.Bef.Res_16 := FALSE;
   Truebwasser_Niv.Bef.Res_17 := FALSE;
   Truebwasser_Niv.Bef.Res_18 := FALSE;
   Truebwasser_Niv.Bef.Res_19 := FALSE;
   Truebwasser_Niv.Bef.Res_20 := FALSE;
   Truebwasser_Niv.Bef.Res_21 := FALSE;
   Truebwasser_Niv.Bef.Res_22 := FALSE;
   Truebwasser_Niv.Bef.Res_23 := FALSE;
   Truebwasser_Niv.Bef.Res_24 := FALSE;
   Truebwasser_Niv.Bef.Res_25 := FALSE;
   Truebwasser_Niv.Bef.Res_26 := FALSE;
   Truebwasser_Niv.Bef.Res_27 := FALSE;
   Truebwasser_Niv.Bef.Res_28 := FALSE;
   Truebwasser_Niv.Bef.Res_29 := FALSE;
   Truebwasser_Niv.Bef.Res_30 := FALSE;
   Truebwasser_Niv.Bef.BF_Quit := FALSE;
   Truebwasser_Niv.MW_Sim := 0.0;
   Truebwasser_DF.Bef.BA_Nrm := FALSE;
   Truebwasser_DF.Bef.BA_Frz := FALSE;
   Truebwasser_DF.Bef.BA_EW := FALSE;
   Truebwasser_DF.Bef.BA_Sim := FALSE;
   Truebwasser_DF.Bef.BA_Wart := FALSE;
   Truebwasser_DF.Bef.Frg_HH := FALSE;
   Truebwasser_DF.Bef.Frg_H := FALSE;
   Truebwasser_DF.Bef.Frg_L := FALSE;
   Truebwasser_DF.Bef.Frg_LL := FALSE;
   Truebwasser_DF.Bef.SB_MW_frz := FALSE;
   Truebwasser_DF.Bef.SB_MW_EW := FALSE;
   Truebwasser_DF.Bef.Res_11 := FALSE;
   Truebwasser_DF.Bef.Res_12 := FALSE;
   Truebwasser_DF.Bef.Res_13 := FALSE;
   Truebwasser_DF.Bef.Res_14 := FALSE;
   Truebwasser_DF.Bef.Res_15 := FALSE;
   Truebwasser_DF.Bef.Res_16 := FALSE;
   Truebwasser_DF.Bef.Res_17 := FALSE;
   Truebwasser_DF.Bef.Res_18 := FALSE;
   Truebwasser_DF.Bef.Res_19 := FALSE;
   Truebwasser_DF.Bef.Res_20 := FALSE;
   Truebwasser_DF.Bef.Res_21 := FALSE;
   Truebwasser_DF.Bef.Res_22 := FALSE;
   Truebwasser_DF.Bef.Res_23 := FALSE;
   Truebwasser_DF.Bef.Res_24 := FALSE;
   Truebwasser_DF.Bef.Res_25 := FALSE;
   Truebwasser_DF.Bef.Res_26 := FALSE;
   Truebwasser_DF.Bef.Res_27 := FALSE;
   Truebwasser_DF.Bef.Res_28 := FALSE;
   Truebwasser_DF.Bef.Res_29 := FALSE;
   Truebwasser_DF.Bef.Res_30 := FALSE;
   Truebwasser_DF.Bef.BF_Quit := FALSE;
   Truebwasser_DF.MW_Sim := 0.0;
   Zulauf_SF_Niv.Bef.BA_Nrm := FALSE;
   Zulauf_SF_Niv.Bef.BA_Frz := FALSE;
   Zulauf_SF_Niv.Bef.BA_EW := FALSE;
   Zulauf_SF_Niv.Bef.BA_Sim := FALSE;
   Zulauf_SF_Niv.Bef.BA_Wart := FALSE;
   Zulauf_SF_Niv.Bef.Frg_HH := FALSE;
   Zulauf_SF_Niv.Bef.Frg_H := FALSE;
   Zulauf_SF_Niv.Bef.Frg_L := FALSE;
   Zulauf_SF_Niv.Bef.Frg_LL := FALSE;
   Zulauf_SF_Niv.Bef.SB_MW_frz := FALSE;
   Zulauf_SF_Niv.Bef.SB_MW_EW := FALSE;
   Zulauf_SF_Niv.Bef.Res_11 := FALSE;
   Zulauf_SF_Niv.Bef.Res_12 := FALSE;
   Zulauf_SF_Niv.Bef.Res_13 := FALSE;
   Zulauf_SF_Niv.Bef.Res_14 := FALSE;
   Zulauf_SF_Niv.Bef.Res_15 := FALSE;
   Zulauf_SF_Niv.Bef.Res_16 := FALSE;
   Zulauf_SF_Niv.Bef.Res_17 := FALSE;
   Zulauf_SF_Niv.Bef.Res_18 := FALSE;
   Zulauf_SF_Niv.Bef.Res_19 := FALSE;
   Zulauf_SF_Niv.Bef.Res_20 := FALSE;
   Zulauf_SF_Niv.Bef.Res_21 := FALSE;
   Zulauf_SF_Niv.Bef.Res_22 := FALSE;
   Zulauf_SF_Niv.Bef.Res_23 := FALSE;
   Zulauf_SF_Niv.Bef.Res_24 := FALSE;
   Zulauf_SF_Niv.Bef.Res_25 := FALSE;
   Zulauf_SF_Niv.Bef.Res_26 := FALSE;
   Zulauf_SF_Niv.Bef.Res_27 := FALSE;
   Zulauf_SF_Niv.Bef.Res_28 := FALSE;
   Zulauf_SF_Niv.Bef.Res_29 := FALSE;
   Zulauf_SF_Niv.Bef.Res_30 := FALSE;
   Zulauf_SF_Niv.Bef.BF_Quit := FALSE;
   Zulauf_SF_Niv.MW_Sim := 0.0;
   Ablauf_NOx.Bef.BA_Nrm := FALSE;
   Ablauf_NOx.Bef.BA_Frz := FALSE;
   Ablauf_NOx.Bef.BA_EW := FALSE;
   Ablauf_NOx.Bef.BA_Sim := FALSE;
   Ablauf_NOx.Bef.BA_Wart := FALSE;
   Ablauf_NOx.Bef.Frg_HH := FALSE;
   Ablauf_NOx.Bef.Frg_H := FALSE;
   Ablauf_NOx.Bef.Frg_L := FALSE;
   Ablauf_NOx.Bef.Frg_LL := FALSE;
   Ablauf_NOx.Bef.SB_MW_frz := FALSE;
   Ablauf_NOx.Bef.SB_MW_EW := FALSE;
   Ablauf_NOx.Bef.Res_11 := FALSE;
   Ablauf_NOx.Bef.Res_12 := FALSE;
   Ablauf_NOx.Bef.Res_13 := FALSE;
   Ablauf_NOx.Bef.Res_14 := FALSE;
   Ablauf_NOx.Bef.Res_15 := FALSE;
   Ablauf_NOx.Bef.Res_16 := FALSE;
   Ablauf_NOx.Bef.Res_17 := FALSE;
   Ablauf_NOx.Bef.Res_18 := FALSE;
   Ablauf_NOx.Bef.Res_19 := FALSE;
   Ablauf_NOx.Bef.Res_20 := FALSE;
   Ablauf_NOx.Bef.Res_21 := FALSE;
   Ablauf_NOx.Bef.Res_22 := FALSE;
   Ablauf_NOx.Bef.Res_23 := FALSE;
   Ablauf_NOx.Bef.Res_24 := FALSE;
   Ablauf_NOx.Bef.Res_25 := FALSE;
   Ablauf_NOx.Bef.Res_26 := FALSE;
   Ablauf_NOx.Bef.Res_27 := FALSE;
   Ablauf_NOx.Bef.Res_28 := FALSE;
   Ablauf_NOx.Bef.Res_29 := FALSE;
   Ablauf_NOx.Bef.Res_30 := FALSE;
   Ablauf_NOx.Bef.BF_Quit := FALSE;
   Ablauf_NOx.MW_Sim := 0.0;
   Ablauf_PO4.Bef.BA_Nrm := FALSE;
   Ablauf_PO4.Bef.BA_Frz := FALSE;
   Ablauf_PO4.Bef.BA_EW := FALSE;
   Ablauf_PO4.Bef.BA_Sim := FALSE;
   Ablauf_PO4.Bef.BA_Wart := FALSE;
   Ablauf_PO4.Bef.Frg_HH := FALSE;
   Ablauf_PO4.Bef.Frg_H := FALSE;
   Ablauf_PO4.Bef.Frg_L := FALSE;
   Ablauf_PO4.Bef.Frg_LL := FALSE;
   Ablauf_PO4.Bef.SB_MW_frz := FALSE;
   Ablauf_PO4.Bef.SB_MW_EW := FALSE;
   Ablauf_PO4.Bef.Res_11 := FALSE;
   Ablauf_PO4.Bef.Res_12 := FALSE;
   Ablauf_PO4.Bef.Res_13 := FALSE;
   Ablauf_PO4.Bef.Res_14 := FALSE;
   Ablauf_PO4.Bef.Res_15 := FALSE;
   Ablauf_PO4.Bef.Res_16 := FALSE;
   Ablauf_PO4.Bef.Res_17 := FALSE;
   Ablauf_PO4.Bef.Res_18 := FALSE;
   Ablauf_PO4.Bef.Res_19 := FALSE;
   Ablauf_PO4.Bef.Res_20 := FALSE;
   Ablauf_PO4.Bef.Res_21 := FALSE;
   Ablauf_PO4.Bef.Res_22 := FALSE;
   Ablauf_PO4.Bef.Res_23 := FALSE;
   Ablauf_PO4.Bef.Res_24 := FALSE;
   Ablauf_PO4.Bef.Res_25 := FALSE;
   Ablauf_PO4.Bef.Res_26 := FALSE;
   Ablauf_PO4.Bef.Res_27 := FALSE;
   Ablauf_PO4.Bef.Res_28 := FALSE;
   Ablauf_PO4.Bef.Res_29 := FALSE;
   Ablauf_PO4.Bef.Res_30 := FALSE;
   Ablauf_PO4.Bef.BF_Quit := FALSE;
   Ablauf_PO4.MW_Sim := 0.0;

END_DATA_BLOCK

DATA_BLOCK "DB116_MW_Prm"
{ S7_Optimized_Access := 'FALSE' }
VERSION : 0.1
   STRUCT
      Zulauf_AR_Niv : "T_MW_PRM";   // Zulauf - Pumpwerk "Alter Rechen" - Niveau
      Zulauf_AR_Temp : "T_MW_PRM";   // Zulauf - Pumpwerk "Alter Rechen" - Temperatur
      Zulauf_AR_DF : "T_MW_PRM";   // Zulauf - Pumpwerk "Alter Rechen" - Durchfluss
      BB1_AS1_SS : "T_MW_PRM";   // Becken 1 - Ablaufschieber 1 - Schieberstellung
      BB1_AS2_SS : "T_MW_PRM";   // Becken 1 - Ablaufschieber 2 - Schieberstellung
      BB2_AS1_SS : "T_MW_PRM";   // Becken 2 - Ablaufschieber 1 - Schieberstellung
      BB2_AS2_SS : "T_MW_PRM";   // Becken 2 - Ablaufschieber 2 - Schieberstellung
      BB1_O2 : "T_MW_PRM";   // Becken 1 - O2-Gehalt
      BB1_Temp : "T_MW_PRM";   // Becken 1 - Temperatur
      BB2_O2 : "T_MW_PRM";   // Becken 2 - O2-Gehalt
      BB2_Temp : "T_MW_PRM";   // Becken 2 - Temperatur
      BB1_DF : "T_MW_PRM";   // Becken 1 - Ablauf - Durchfluss
      BB2_DF : "T_MW_PRM";   // Becken 2 - Ablauf - Durchfluss
      Zulauf_Niv : "T_MW_PRM";   // Zulauf - Vorlagebehälter - Niveau
      Zulauf_DF : "T_MW_PRM";   // Zulauf - Rechen - Durchfluss
      Verteiler_pH : "T_MW_PRM";   // Zulauf - Verteiler - pH-Wert
      Verteiler_O2 : "T_MW_PRM";   // Zulauf - Verteiler  - O2-Gehalt
      Verteiler_Temp : "T_MW_PRM";   // Zulauf - Verteiler - Temperatur
      BB_UeSS_DF : "T_MW_PRM";   // Becken 1+2 - Ablauf ÜSS - Durchfluss
      Ablauf_DF : "T_MW_PRM";   // Ablauf - Durchfluss
      Ablauf_pH : "T_MW_PRM";   // Ablauf - pH-Wert
      Ablauf_O2 : "T_MW_PRM";   // Ablauf - O2-Gehalt
      Ablauf_Temp : "T_MW_PRM";   // Ablauf - Temperatur
      Schlamm_ED_Niv : "T_MW_PRM";   // Schlamm - Eindicker - Niveau
      Schlamm_Besch_Niv : "T_MW_PRM";   // Schlamm - Beschickung - Niveau
      Schlamm_Besch_DF : "T_MW_PRM";   // Schlamm - Beschickung - Durchfluss
      Truebwasser_Niv : "T_MW_PRM";   // Trübwasserpumpwerk - Niveau
      Truebwasser_DF : "T_MW_PRM";   // Trübwasserpumpwerk - Durchfluss
      Zulauf_SF_Niv : "T_MW_PRM";   // Zulauf - Sandfang - Niveau
      Ablauf_NOx : "T_MW_PRM";   // Ablauf - Dortmundbrunnen - Nitratmessung
      Ablauf_PO4 : "T_MW_PRM";   // Ablauf - Dortmundbrunnen - Phosphatmessung
      Umwelt_WG : "T_MW_PRM";   // Wetterstation - Windgeschwindigkeit
      Umwelt_WR : "T_MW_PRM";   // Wetterstation - Windrichtung
      Umwelt_LDr : "T_MW_PRM";   // Wetterstation - Luftdruck
      Umwelt_LF : "T_MW_PRM";   // Wetterstation - Luftfeuchtigkeit
      Umwelt_T : "T_MW_PRM";   // Wetterstation - Temperatur
      Ablauf_LF : "T_MW_PRM";   // Ablauf - Leitfähigkeit
   END_STRUCT;


BEGIN
   Zulauf_AR_Niv.Konfig.Peri := TRUE;
   Zulauf_AR_Niv.Konfig.PW := FALSE;
   Zulauf_AR_Niv.Konfig.Peri_0_20mA := FALSE;
   Zulauf_AR_Niv.Konfig.Peri_4_20mA := TRUE;
   Zulauf_AR_Niv.Konfig.Peri_PT100 := FALSE;
   Zulauf_AR_Niv.Konfig.GW_Delta := FALSE;
   Zulauf_AR_Niv.Konfig.Res_6 := FALSE;
   Zulauf_AR_Niv.Konfig.Res_7 := FALSE;
   Zulauf_AR_Niv.Konfig.Res_8 := FALSE;
   Zulauf_AR_Niv.Konfig.Res_9 := FALSE;
   Zulauf_AR_Niv.Konfig.Res_10 := FALSE;
   Zulauf_AR_Niv.Konfig.Res_11 := FALSE;
   Zulauf_AR_Niv.Konfig.Res_12 := FALSE;
   Zulauf_AR_Niv.Konfig.Res_13 := FALSE;
   Zulauf_AR_Niv.Konfig.Res_14 := FALSE;
   Zulauf_AR_Niv.Konfig.Res_15 := FALSE;
   Zulauf_AR_Niv.Konfig.Res_16 := FALSE;
   Zulauf_AR_Niv.Konfig.Res_17 := FALSE;
   Zulauf_AR_Niv.Konfig.Res_18 := FALSE;
   Zulauf_AR_Niv.Konfig.Res_19 := FALSE;
   Zulauf_AR_Niv.Konfig.Res_20 := FALSE;
   Zulauf_AR_Niv.Konfig.Res_21 := FALSE;
   Zulauf_AR_Niv.Konfig.Res_22 := FALSE;
   Zulauf_AR_Niv.Konfig.Res_23 := FALSE;
   Zulauf_AR_Niv.Konfig.Res_24 := FALSE;
   Zulauf_AR_Niv.Konfig.Res_25 := FALSE;
   Zulauf_AR_Niv.Konfig.Res_26 := FALSE;
   Zulauf_AR_Niv.Konfig.Res_27 := FALSE;
   Zulauf_AR_Niv.Konfig.Res_28 := FALSE;
   Zulauf_AR_Niv.Konfig.Res_29 := FALSE;
   Zulauf_AR_Niv.Konfig.Res_30 := FALSE;
   Zulauf_AR_Niv.Konfig.Res_31 := FALSE;
   Zulauf_AR_Niv.MW_EW := 0.0;
   Zulauf_AR_Niv.MW_OG := 100.0;
   Zulauf_AR_Niv.MW_UG := 0.0;
   Zulauf_AR_Niv.GW_HH := 100.0;
   Zulauf_AR_Niv.GW_H := 100.0;
   Zulauf_AR_Niv.GW_L := 0.0;
   Zulauf_AR_Niv.GW_LL := 0.0;
   Zulauf_AR_Niv.GW_Hyst := 1.0;
   Zulauf_AR_Niv.VZ_St := 5;
   Zulauf_AR_Niv.VZ_Ex := 15;
   Zulauf_AR_Niv.MW_Avg := 5;
   Zulauf_AR_Temp.Konfig.Peri := TRUE;
   Zulauf_AR_Temp.Konfig.PW := FALSE;
   Zulauf_AR_Temp.Konfig.Peri_0_20mA := FALSE;
   Zulauf_AR_Temp.Konfig.Peri_4_20mA := TRUE;
   Zulauf_AR_Temp.Konfig.Peri_PT100 := FALSE;
   Zulauf_AR_Temp.Konfig.GW_Delta := FALSE;
   Zulauf_AR_Temp.Konfig.Res_6 := FALSE;
   Zulauf_AR_Temp.Konfig.Res_7 := FALSE;
   Zulauf_AR_Temp.Konfig.Res_8 := FALSE;
   Zulauf_AR_Temp.Konfig.Res_9 := FALSE;
   Zulauf_AR_Temp.Konfig.Res_10 := FALSE;
   Zulauf_AR_Temp.Konfig.Res_11 := FALSE;
   Zulauf_AR_Temp.Konfig.Res_12 := FALSE;
   Zulauf_AR_Temp.Konfig.Res_13 := FALSE;
   Zulauf_AR_Temp.Konfig.Res_14 := FALSE;
   Zulauf_AR_Temp.Konfig.Res_15 := FALSE;
   Zulauf_AR_Temp.Konfig.Res_16 := FALSE;
   Zulauf_AR_Temp.Konfig.Res_17 := FALSE;
   Zulauf_AR_Temp.Konfig.Res_18 := FALSE;
   Zulauf_AR_Temp.Konfig.Res_19 := FALSE;
   Zulauf_AR_Temp.Konfig.Res_20 := FALSE;
   Zulauf_AR_Temp.Konfig.Res_21 := FALSE;
   Zulauf_AR_Temp.Konfig.Res_22 := FALSE;
   Zulauf_AR_Temp.Konfig.Res_23 := FALSE;
   Zulauf_AR_Temp.Konfig.Res_24 := FALSE;
   Zulauf_AR_Temp.Konfig.Res_25 := FALSE;
   Zulauf_AR_Temp.Konfig.Res_26 := FALSE;
   Zulauf_AR_Temp.Konfig.Res_27 := FALSE;
   Zulauf_AR_Temp.Konfig.Res_28 := FALSE;
   Zulauf_AR_Temp.Konfig.Res_29 := FALSE;
   Zulauf_AR_Temp.Konfig.Res_30 := FALSE;
   Zulauf_AR_Temp.Konfig.Res_31 := FALSE;
   Zulauf_AR_Temp.MW_EW := 0.0;
   Zulauf_AR_Temp.MW_OG := 50.0;
   Zulauf_AR_Temp.MW_UG := 0.0;
   Zulauf_AR_Temp.GW_HH := 50.0;
   Zulauf_AR_Temp.GW_H := 50.0;
   Zulauf_AR_Temp.GW_L := 0.0;
   Zulauf_AR_Temp.GW_LL := 0.0;
   Zulauf_AR_Temp.GW_Hyst := 1.0;
   Zulauf_AR_Temp.VZ_St := 5;
   Zulauf_AR_Temp.VZ_Ex := 3;
   Zulauf_AR_Temp.MW_Avg := 3;
   Zulauf_AR_DF.Konfig.Peri := TRUE;
   Zulauf_AR_DF.Konfig.PW := FALSE;
   Zulauf_AR_DF.Konfig.Peri_0_20mA := FALSE;
   Zulauf_AR_DF.Konfig.Peri_4_20mA := TRUE;
   Zulauf_AR_DF.Konfig.Peri_PT100 := FALSE;
   Zulauf_AR_DF.Konfig.GW_Delta := FALSE;
   Zulauf_AR_DF.Konfig.Res_6 := FALSE;
   Zulauf_AR_DF.Konfig.Res_7 := FALSE;
   Zulauf_AR_DF.Konfig.Res_8 := FALSE;
   Zulauf_AR_DF.Konfig.Res_9 := FALSE;
   Zulauf_AR_DF.Konfig.Res_10 := FALSE;
   Zulauf_AR_DF.Konfig.Res_11 := FALSE;
   Zulauf_AR_DF.Konfig.Res_12 := FALSE;
   Zulauf_AR_DF.Konfig.Res_13 := FALSE;
   Zulauf_AR_DF.Konfig.Res_14 := FALSE;
   Zulauf_AR_DF.Konfig.Res_15 := FALSE;
   Zulauf_AR_DF.Konfig.Res_16 := FALSE;
   Zulauf_AR_DF.Konfig.Res_17 := FALSE;
   Zulauf_AR_DF.Konfig.Res_18 := FALSE;
   Zulauf_AR_DF.Konfig.Res_19 := FALSE;
   Zulauf_AR_DF.Konfig.Res_20 := FALSE;
   Zulauf_AR_DF.Konfig.Res_21 := FALSE;
   Zulauf_AR_DF.Konfig.Res_22 := FALSE;
   Zulauf_AR_DF.Konfig.Res_23 := FALSE;
   Zulauf_AR_DF.Konfig.Res_24 := FALSE;
   Zulauf_AR_DF.Konfig.Res_25 := FALSE;
   Zulauf_AR_DF.Konfig.Res_26 := FALSE;
   Zulauf_AR_DF.Konfig.Res_27 := FALSE;
   Zulauf_AR_DF.Konfig.Res_28 := FALSE;
   Zulauf_AR_DF.Konfig.Res_29 := FALSE;
   Zulauf_AR_DF.Konfig.Res_30 := FALSE;
   Zulauf_AR_DF.Konfig.Res_31 := FALSE;
   Zulauf_AR_DF.MW_EW := 0.0;
   Zulauf_AR_DF.MW_OG := 20.0;
   Zulauf_AR_DF.MW_UG := 0.0;
   Zulauf_AR_DF.GW_HH := 20.0;
   Zulauf_AR_DF.GW_H := 20.0;
   Zulauf_AR_DF.GW_L := 0.0;
   Zulauf_AR_DF.GW_LL := 0.0;
   Zulauf_AR_DF.GW_Hyst := 1.0;
   Zulauf_AR_DF.VZ_St := 5;
   Zulauf_AR_DF.VZ_Ex := 15;
   Zulauf_AR_DF.MW_Avg := 3;
   BB1_AS1_SS.Konfig.Peri := TRUE;
   BB1_AS1_SS.Konfig.PW := FALSE;
   BB1_AS1_SS.Konfig.Peri_0_20mA := FALSE;
   BB1_AS1_SS.Konfig.Peri_4_20mA := TRUE;
   BB1_AS1_SS.Konfig.Peri_PT100 := FALSE;
   BB1_AS1_SS.Konfig.GW_Delta := FALSE;
   BB1_AS1_SS.Konfig.Res_6 := FALSE;
   BB1_AS1_SS.Konfig.Res_7 := FALSE;
   BB1_AS1_SS.Konfig.Res_8 := FALSE;
   BB1_AS1_SS.Konfig.Res_9 := FALSE;
   BB1_AS1_SS.Konfig.Res_10 := FALSE;
   BB1_AS1_SS.Konfig.Res_11 := FALSE;
   BB1_AS1_SS.Konfig.Res_12 := FALSE;
   BB1_AS1_SS.Konfig.Res_13 := FALSE;
   BB1_AS1_SS.Konfig.Res_14 := FALSE;
   BB1_AS1_SS.Konfig.Res_15 := FALSE;
   BB1_AS1_SS.Konfig.Res_16 := FALSE;
   BB1_AS1_SS.Konfig.Res_17 := FALSE;
   BB1_AS1_SS.Konfig.Res_18 := FALSE;
   BB1_AS1_SS.Konfig.Res_19 := FALSE;
   BB1_AS1_SS.Konfig.Res_20 := FALSE;
   BB1_AS1_SS.Konfig.Res_21 := FALSE;
   BB1_AS1_SS.Konfig.Res_22 := FALSE;
   BB1_AS1_SS.Konfig.Res_23 := FALSE;
   BB1_AS1_SS.Konfig.Res_24 := FALSE;
   BB1_AS1_SS.Konfig.Res_25 := FALSE;
   BB1_AS1_SS.Konfig.Res_26 := FALSE;
   BB1_AS1_SS.Konfig.Res_27 := FALSE;
   BB1_AS1_SS.Konfig.Res_28 := FALSE;
   BB1_AS1_SS.Konfig.Res_29 := FALSE;
   BB1_AS1_SS.Konfig.Res_30 := FALSE;
   BB1_AS1_SS.Konfig.Res_31 := FALSE;
   BB1_AS1_SS.MW_EW := 0.0;
   BB1_AS1_SS.MW_OG := 100.0;
   BB1_AS1_SS.MW_UG := 0.0;
   BB1_AS1_SS.GW_HH := 100.0;
   BB1_AS1_SS.GW_H := 100.0;
   BB1_AS1_SS.GW_L := 0.0;
   BB1_AS1_SS.GW_LL := 0.0;
   BB1_AS1_SS.GW_Hyst := 1.0;
   BB1_AS1_SS.VZ_St := 5;
   BB1_AS1_SS.VZ_Ex := 15;
   BB1_AS1_SS.MW_Avg := 30;
   BB1_AS2_SS.Konfig.Peri := TRUE;
   BB1_AS2_SS.Konfig.PW := FALSE;
   BB1_AS2_SS.Konfig.Peri_0_20mA := FALSE;
   BB1_AS2_SS.Konfig.Peri_4_20mA := TRUE;
   BB1_AS2_SS.Konfig.Peri_PT100 := FALSE;
   BB1_AS2_SS.Konfig.GW_Delta := FALSE;
   BB1_AS2_SS.Konfig.Res_6 := FALSE;
   BB1_AS2_SS.Konfig.Res_7 := FALSE;
   BB1_AS2_SS.Konfig.Res_8 := FALSE;
   BB1_AS2_SS.Konfig.Res_9 := FALSE;
   BB1_AS2_SS.Konfig.Res_10 := FALSE;
   BB1_AS2_SS.Konfig.Res_11 := FALSE;
   BB1_AS2_SS.Konfig.Res_12 := FALSE;
   BB1_AS2_SS.Konfig.Res_13 := FALSE;
   BB1_AS2_SS.Konfig.Res_14 := FALSE;
   BB1_AS2_SS.Konfig.Res_15 := FALSE;
   BB1_AS2_SS.Konfig.Res_16 := FALSE;
   BB1_AS2_SS.Konfig.Res_17 := FALSE;
   BB1_AS2_SS.Konfig.Res_18 := FALSE;
   BB1_AS2_SS.Konfig.Res_19 := FALSE;
   BB1_AS2_SS.Konfig.Res_20 := FALSE;
   BB1_AS2_SS.Konfig.Res_21 := FALSE;
   BB1_AS2_SS.Konfig.Res_22 := FALSE;
   BB1_AS2_SS.Konfig.Res_23 := FALSE;
   BB1_AS2_SS.Konfig.Res_24 := FALSE;
   BB1_AS2_SS.Konfig.Res_25 := FALSE;
   BB1_AS2_SS.Konfig.Res_26 := FALSE;
   BB1_AS2_SS.Konfig.Res_27 := FALSE;
   BB1_AS2_SS.Konfig.Res_28 := FALSE;
   BB1_AS2_SS.Konfig.Res_29 := FALSE;
   BB1_AS2_SS.Konfig.Res_30 := FALSE;
   BB1_AS2_SS.Konfig.Res_31 := FALSE;
   BB1_AS2_SS.MW_EW := 0.0;
   BB1_AS2_SS.MW_OG := 100.0;
   BB1_AS2_SS.MW_UG := 0.0;
   BB1_AS2_SS.GW_HH := 100.0;
   BB1_AS2_SS.GW_H := 100.0;
   BB1_AS2_SS.GW_L := 0.0;
   BB1_AS2_SS.GW_LL := 0.0;
   BB1_AS2_SS.GW_Hyst := 1.0;
   BB1_AS2_SS.VZ_St := 5;
   BB1_AS2_SS.VZ_Ex := 15;
   BB1_AS2_SS.MW_Avg := 10;
   BB2_AS1_SS.Konfig.Peri := TRUE;
   BB2_AS1_SS.Konfig.PW := FALSE;
   BB2_AS1_SS.Konfig.Peri_0_20mA := FALSE;
   BB2_AS1_SS.Konfig.Peri_4_20mA := TRUE;
   BB2_AS1_SS.Konfig.Peri_PT100 := FALSE;
   BB2_AS1_SS.Konfig.GW_Delta := FALSE;
   BB2_AS1_SS.Konfig.Res_6 := FALSE;
   BB2_AS1_SS.Konfig.Res_7 := FALSE;
   BB2_AS1_SS.Konfig.Res_8 := FALSE;
   BB2_AS1_SS.Konfig.Res_9 := FALSE;
   BB2_AS1_SS.Konfig.Res_10 := FALSE;
   BB2_AS1_SS.Konfig.Res_11 := FALSE;
   BB2_AS1_SS.Konfig.Res_12 := FALSE;
   BB2_AS1_SS.Konfig.Res_13 := FALSE;
   BB2_AS1_SS.Konfig.Res_14 := FALSE;
   BB2_AS1_SS.Konfig.Res_15 := FALSE;
   BB2_AS1_SS.Konfig.Res_16 := FALSE;
   BB2_AS1_SS.Konfig.Res_17 := FALSE;
   BB2_AS1_SS.Konfig.Res_18 := FALSE;
   BB2_AS1_SS.Konfig.Res_19 := FALSE;
   BB2_AS1_SS.Konfig.Res_20 := FALSE;
   BB2_AS1_SS.Konfig.Res_21 := FALSE;
   BB2_AS1_SS.Konfig.Res_22 := FALSE;
   BB2_AS1_SS.Konfig.Res_23 := FALSE;
   BB2_AS1_SS.Konfig.Res_24 := FALSE;
   BB2_AS1_SS.Konfig.Res_25 := FALSE;
   BB2_AS1_SS.Konfig.Res_26 := FALSE;
   BB2_AS1_SS.Konfig.Res_27 := FALSE;
   BB2_AS1_SS.Konfig.Res_28 := FALSE;
   BB2_AS1_SS.Konfig.Res_29 := FALSE;
   BB2_AS1_SS.Konfig.Res_30 := FALSE;
   BB2_AS1_SS.Konfig.Res_31 := FALSE;
   BB2_AS1_SS.MW_EW := 0.0;
   BB2_AS1_SS.MW_OG := 100.0;
   BB2_AS1_SS.MW_UG := 0.0;
   BB2_AS1_SS.GW_HH := 100.0;
   BB2_AS1_SS.GW_H := 100.0;
   BB2_AS1_SS.GW_L := 0.0;
   BB2_AS1_SS.GW_LL := 0.0;
   BB2_AS1_SS.GW_Hyst := 1.0;
   BB2_AS1_SS.VZ_St := 5;
   BB2_AS1_SS.VZ_Ex := 15;
   BB2_AS1_SS.MW_Avg := 10;
   BB2_AS2_SS.Konfig.Peri := TRUE;
   BB2_AS2_SS.Konfig.PW := FALSE;
   BB2_AS2_SS.Konfig.Peri_0_20mA := FALSE;
   BB2_AS2_SS.Konfig.Peri_4_20mA := TRUE;
   BB2_AS2_SS.Konfig.Peri_PT100 := FALSE;
   BB2_AS2_SS.Konfig.GW_Delta := FALSE;
   BB2_AS2_SS.Konfig.Res_6 := FALSE;
   BB2_AS2_SS.Konfig.Res_7 := FALSE;
   BB2_AS2_SS.Konfig.Res_8 := FALSE;
   BB2_AS2_SS.Konfig.Res_9 := FALSE;
   BB2_AS2_SS.Konfig.Res_10 := FALSE;
   BB2_AS2_SS.Konfig.Res_11 := FALSE;
   BB2_AS2_SS.Konfig.Res_12 := FALSE;
   BB2_AS2_SS.Konfig.Res_13 := FALSE;
   BB2_AS2_SS.Konfig.Res_14 := FALSE;
   BB2_AS2_SS.Konfig.Res_15 := FALSE;
   BB2_AS2_SS.Konfig.Res_16 := FALSE;
   BB2_AS2_SS.Konfig.Res_17 := FALSE;
   BB2_AS2_SS.Konfig.Res_18 := FALSE;
   BB2_AS2_SS.Konfig.Res_19 := FALSE;
   BB2_AS2_SS.Konfig.Res_20 := FALSE;
   BB2_AS2_SS.Konfig.Res_21 := FALSE;
   BB2_AS2_SS.Konfig.Res_22 := FALSE;
   BB2_AS2_SS.Konfig.Res_23 := FALSE;
   BB2_AS2_SS.Konfig.Res_24 := FALSE;
   BB2_AS2_SS.Konfig.Res_25 := FALSE;
   BB2_AS2_SS.Konfig.Res_26 := FALSE;
   BB2_AS2_SS.Konfig.Res_27 := FALSE;
   BB2_AS2_SS.Konfig.Res_28 := FALSE;
   BB2_AS2_SS.Konfig.Res_29 := FALSE;
   BB2_AS2_SS.Konfig.Res_30 := FALSE;
   BB2_AS2_SS.Konfig.Res_31 := FALSE;
   BB2_AS2_SS.MW_EW := 0.0;
   BB2_AS2_SS.MW_OG := 100.0;
   BB2_AS2_SS.MW_UG := 0.0;
   BB2_AS2_SS.GW_HH := 100.0;
   BB2_AS2_SS.GW_H := 100.0;
   BB2_AS2_SS.GW_L := 0.0;
   BB2_AS2_SS.GW_LL := 0.0;
   BB2_AS2_SS.GW_Hyst := 1.0;
   BB2_AS2_SS.VZ_St := 5;
   BB2_AS2_SS.VZ_Ex := 15;
   BB2_AS2_SS.MW_Avg := 10;
   BB1_O2.Konfig.Peri := TRUE;
   BB1_O2.Konfig.PW := FALSE;
   BB1_O2.Konfig.Peri_0_20mA := FALSE;
   BB1_O2.Konfig.Peri_4_20mA := TRUE;
   BB1_O2.Konfig.Peri_PT100 := FALSE;
   BB1_O2.Konfig.GW_Delta := FALSE;
   BB1_O2.Konfig.Res_6 := FALSE;
   BB1_O2.Konfig.Res_7 := FALSE;
   BB1_O2.Konfig.Res_8 := FALSE;
   BB1_O2.Konfig.Res_9 := FALSE;
   BB1_O2.Konfig.Res_10 := FALSE;
   BB1_O2.Konfig.Res_11 := FALSE;
   BB1_O2.Konfig.Res_12 := FALSE;
   BB1_O2.Konfig.Res_13 := FALSE;
   BB1_O2.Konfig.Res_14 := FALSE;
   BB1_O2.Konfig.Res_15 := FALSE;
   BB1_O2.Konfig.Res_16 := FALSE;
   BB1_O2.Konfig.Res_17 := FALSE;
   BB1_O2.Konfig.Res_18 := FALSE;
   BB1_O2.Konfig.Res_19 := FALSE;
   BB1_O2.Konfig.Res_20 := FALSE;
   BB1_O2.Konfig.Res_21 := FALSE;
   BB1_O2.Konfig.Res_22 := FALSE;
   BB1_O2.Konfig.Res_23 := FALSE;
   BB1_O2.Konfig.Res_24 := FALSE;
   BB1_O2.Konfig.Res_25 := FALSE;
   BB1_O2.Konfig.Res_26 := FALSE;
   BB1_O2.Konfig.Res_27 := FALSE;
   BB1_O2.Konfig.Res_28 := FALSE;
   BB1_O2.Konfig.Res_29 := FALSE;
   BB1_O2.Konfig.Res_30 := FALSE;
   BB1_O2.Konfig.Res_31 := FALSE;
   BB1_O2.MW_EW := 0.0;
   BB1_O2.MW_OG := 10.0;
   BB1_O2.MW_UG := 0.0;
   BB1_O2.GW_HH := 10.0;
   BB1_O2.GW_H := 10.0;
   BB1_O2.GW_L := 0.4;
   BB1_O2.GW_LL := 0.4;
   BB1_O2.GW_Hyst := 0.1;
   BB1_O2.VZ_St := 5;
   BB1_O2.VZ_Ex := 7200;
   BB1_O2.MW_Avg := 30;
   BB1_Temp.Konfig.Peri := TRUE;
   BB1_Temp.Konfig.PW := FALSE;
   BB1_Temp.Konfig.Peri_0_20mA := FALSE;
   BB1_Temp.Konfig.Peri_4_20mA := TRUE;
   BB1_Temp.Konfig.Peri_PT100 := FALSE;
   BB1_Temp.Konfig.GW_Delta := FALSE;
   BB1_Temp.Konfig.Res_6 := FALSE;
   BB1_Temp.Konfig.Res_7 := FALSE;
   BB1_Temp.Konfig.Res_8 := FALSE;
   BB1_Temp.Konfig.Res_9 := FALSE;
   BB1_Temp.Konfig.Res_10 := FALSE;
   BB1_Temp.Konfig.Res_11 := FALSE;
   BB1_Temp.Konfig.Res_12 := FALSE;
   BB1_Temp.Konfig.Res_13 := FALSE;
   BB1_Temp.Konfig.Res_14 := FALSE;
   BB1_Temp.Konfig.Res_15 := FALSE;
   BB1_Temp.Konfig.Res_16 := FALSE;
   BB1_Temp.Konfig.Res_17 := FALSE;
   BB1_Temp.Konfig.Res_18 := FALSE;
   BB1_Temp.Konfig.Res_19 := FALSE;
   BB1_Temp.Konfig.Res_20 := FALSE;
   BB1_Temp.Konfig.Res_21 := FALSE;
   BB1_Temp.Konfig.Res_22 := FALSE;
   BB1_Temp.Konfig.Res_23 := FALSE;
   BB1_Temp.Konfig.Res_24 := FALSE;
   BB1_Temp.Konfig.Res_25 := FALSE;
   BB1_Temp.Konfig.Res_26 := FALSE;
   BB1_Temp.Konfig.Res_27 := FALSE;
   BB1_Temp.Konfig.Res_28 := FALSE;
   BB1_Temp.Konfig.Res_29 := FALSE;
   BB1_Temp.Konfig.Res_30 := FALSE;
   BB1_Temp.Konfig.Res_31 := FALSE;
   BB1_Temp.MW_EW := 0.0;
   BB1_Temp.MW_OG := 50.0;
   BB1_Temp.MW_UG := 0.0;
   BB1_Temp.GW_HH := 50.0;
   BB1_Temp.GW_H := 50.0;
   BB1_Temp.GW_L := 0.0;
   BB1_Temp.GW_LL := 0.0;
   BB1_Temp.GW_Hyst := 1.0;
   BB1_Temp.VZ_St := 5;
   BB1_Temp.VZ_Ex := 15;
   BB1_Temp.MW_Avg := 30;
   BB2_O2.Konfig.Peri := TRUE;
   BB2_O2.Konfig.PW := FALSE;
   BB2_O2.Konfig.Peri_0_20mA := FALSE;
   BB2_O2.Konfig.Peri_4_20mA := TRUE;
   BB2_O2.Konfig.Peri_PT100 := FALSE;
   BB2_O2.Konfig.GW_Delta := FALSE;
   BB2_O2.Konfig.Res_6 := FALSE;
   BB2_O2.Konfig.Res_7 := FALSE;
   BB2_O2.Konfig.Res_8 := FALSE;
   BB2_O2.Konfig.Res_9 := FALSE;
   BB2_O2.Konfig.Res_10 := FALSE;
   BB2_O2.Konfig.Res_11 := FALSE;
   BB2_O2.Konfig.Res_12 := FALSE;
   BB2_O2.Konfig.Res_13 := FALSE;
   BB2_O2.Konfig.Res_14 := FALSE;
   BB2_O2.Konfig.Res_15 := FALSE;
   BB2_O2.Konfig.Res_16 := FALSE;
   BB2_O2.Konfig.Res_17 := FALSE;
   BB2_O2.Konfig.Res_18 := FALSE;
   BB2_O2.Konfig.Res_19 := FALSE;
   BB2_O2.Konfig.Res_20 := FALSE;
   BB2_O2.Konfig.Res_21 := FALSE;
   BB2_O2.Konfig.Res_22 := FALSE;
   BB2_O2.Konfig.Res_23 := FALSE;
   BB2_O2.Konfig.Res_24 := FALSE;
   BB2_O2.Konfig.Res_25 := FALSE;
   BB2_O2.Konfig.Res_26 := FALSE;
   BB2_O2.Konfig.Res_27 := FALSE;
   BB2_O2.Konfig.Res_28 := FALSE;
   BB2_O2.Konfig.Res_29 := FALSE;
   BB2_O2.Konfig.Res_30 := FALSE;
   BB2_O2.Konfig.Res_31 := FALSE;
   BB2_O2.MW_EW := 0.0;
   BB2_O2.MW_OG := 10.0;
   BB2_O2.MW_UG := 0.0;
   BB2_O2.GW_HH := 10.0;
   BB2_O2.GW_H := 10.0;
   BB2_O2.GW_L := 0.4;
   BB2_O2.GW_LL := 0.2;
   BB2_O2.GW_Hyst := 0.1;
   BB2_O2.VZ_St := 5;
   BB2_O2.VZ_Ex := 7200;
   BB2_O2.MW_Avg := 30;
   BB2_Temp.Konfig.Peri := TRUE;
   BB2_Temp.Konfig.PW := FALSE;
   BB2_Temp.Konfig.Peri_0_20mA := FALSE;
   BB2_Temp.Konfig.Peri_4_20mA := TRUE;
   BB2_Temp.Konfig.Peri_PT100 := FALSE;
   BB2_Temp.Konfig.GW_Delta := FALSE;
   BB2_Temp.Konfig.Res_6 := FALSE;
   BB2_Temp.Konfig.Res_7 := FALSE;
   BB2_Temp.Konfig.Res_8 := FALSE;
   BB2_Temp.Konfig.Res_9 := FALSE;
   BB2_Temp.Konfig.Res_10 := FALSE;
   BB2_Temp.Konfig.Res_11 := FALSE;
   BB2_Temp.Konfig.Res_12 := FALSE;
   BB2_Temp.Konfig.Res_13 := FALSE;
   BB2_Temp.Konfig.Res_14 := FALSE;
   BB2_Temp.Konfig.Res_15 := FALSE;
   BB2_Temp.Konfig.Res_16 := FALSE;
   BB2_Temp.Konfig.Res_17 := FALSE;
   BB2_Temp.Konfig.Res_18 := FALSE;
   BB2_Temp.Konfig.Res_19 := FALSE;
   BB2_Temp.Konfig.Res_20 := FALSE;
   BB2_Temp.Konfig.Res_21 := FALSE;
   BB2_Temp.Konfig.Res_22 := FALSE;
   BB2_Temp.Konfig.Res_23 := FALSE;
   BB2_Temp.Konfig.Res_24 := FALSE;
   BB2_Temp.Konfig.Res_25 := FALSE;
   BB2_Temp.Konfig.Res_26 := FALSE;
   BB2_Temp.Konfig.Res_27 := FALSE;
   BB2_Temp.Konfig.Res_28 := FALSE;
   BB2_Temp.Konfig.Res_29 := FALSE;
   BB2_Temp.Konfig.Res_30 := FALSE;
   BB2_Temp.Konfig.Res_31 := FALSE;
   BB2_Temp.MW_EW := 0.0;
   BB2_Temp.MW_OG := 50.0;
   BB2_Temp.MW_UG := 0.0;
   BB2_Temp.GW_HH := 50.0;
   BB2_Temp.GW_H := 50.0;
   BB2_Temp.GW_L := 0.0;
   BB2_Temp.GW_LL := 0.0;
   BB2_Temp.GW_Hyst := 1.0;
   BB2_Temp.VZ_St := 5;
   BB2_Temp.VZ_Ex := 15;
   BB2_Temp.MW_Avg := 30;
   BB1_DF.Konfig.Peri := TRUE;
   BB1_DF.Konfig.PW := FALSE;
   BB1_DF.Konfig.Peri_0_20mA := FALSE;
   BB1_DF.Konfig.Peri_4_20mA := TRUE;
   BB1_DF.Konfig.Peri_PT100 := FALSE;
   BB1_DF.Konfig.GW_Delta := FALSE;
   BB1_DF.Konfig.Res_6 := FALSE;
   BB1_DF.Konfig.Res_7 := FALSE;
   BB1_DF.Konfig.Res_8 := FALSE;
   BB1_DF.Konfig.Res_9 := FALSE;
   BB1_DF.Konfig.Res_10 := FALSE;
   BB1_DF.Konfig.Res_11 := FALSE;
   BB1_DF.Konfig.Res_12 := FALSE;
   BB1_DF.Konfig.Res_13 := FALSE;
   BB1_DF.Konfig.Res_14 := FALSE;
   BB1_DF.Konfig.Res_15 := FALSE;
   BB1_DF.Konfig.Res_16 := FALSE;
   BB1_DF.Konfig.Res_17 := FALSE;
   BB1_DF.Konfig.Res_18 := FALSE;
   BB1_DF.Konfig.Res_19 := FALSE;
   BB1_DF.Konfig.Res_20 := FALSE;
   BB1_DF.Konfig.Res_21 := FALSE;
   BB1_DF.Konfig.Res_22 := FALSE;
   BB1_DF.Konfig.Res_23 := FALSE;
   BB1_DF.Konfig.Res_24 := FALSE;
   BB1_DF.Konfig.Res_25 := FALSE;
   BB1_DF.Konfig.Res_26 := FALSE;
   BB1_DF.Konfig.Res_27 := FALSE;
   BB1_DF.Konfig.Res_28 := FALSE;
   BB1_DF.Konfig.Res_29 := FALSE;
   BB1_DF.Konfig.Res_30 := FALSE;
   BB1_DF.Konfig.Res_31 := FALSE;
   BB1_DF.MW_EW := 0.0;
   BB1_DF.MW_OG := 100.0;
   BB1_DF.MW_UG := 0.0;
   BB1_DF.GW_HH := 100.0;
   BB1_DF.GW_H := 100.0;
   BB1_DF.GW_L := 0.0;
   BB1_DF.GW_LL := 0.0;
   BB1_DF.GW_Hyst := 1.0;
   BB1_DF.VZ_St := 5;
   BB1_DF.VZ_Ex := 15;
   BB1_DF.MW_Avg := 10;
   BB2_DF.Konfig.Peri := TRUE;
   BB2_DF.Konfig.PW := FALSE;
   BB2_DF.Konfig.Peri_0_20mA := FALSE;
   BB2_DF.Konfig.Peri_4_20mA := TRUE;
   BB2_DF.Konfig.Peri_PT100 := FALSE;
   BB2_DF.Konfig.GW_Delta := FALSE;
   BB2_DF.Konfig.Res_6 := FALSE;
   BB2_DF.Konfig.Res_7 := FALSE;
   BB2_DF.Konfig.Res_8 := FALSE;
   BB2_DF.Konfig.Res_9 := FALSE;
   BB2_DF.Konfig.Res_10 := FALSE;
   BB2_DF.Konfig.Res_11 := FALSE;
   BB2_DF.Konfig.Res_12 := FALSE;
   BB2_DF.Konfig.Res_13 := FALSE;
   BB2_DF.Konfig.Res_14 := FALSE;
   BB2_DF.Konfig.Res_15 := FALSE;
   BB2_DF.Konfig.Res_16 := FALSE;
   BB2_DF.Konfig.Res_17 := FALSE;
   BB2_DF.Konfig.Res_18 := FALSE;
   BB2_DF.Konfig.Res_19 := FALSE;
   BB2_DF.Konfig.Res_20 := FALSE;
   BB2_DF.Konfig.Res_21 := FALSE;
   BB2_DF.Konfig.Res_22 := FALSE;
   BB2_DF.Konfig.Res_23 := FALSE;
   BB2_DF.Konfig.Res_24 := FALSE;
   BB2_DF.Konfig.Res_25 := FALSE;
   BB2_DF.Konfig.Res_26 := FALSE;
   BB2_DF.Konfig.Res_27 := FALSE;
   BB2_DF.Konfig.Res_28 := FALSE;
   BB2_DF.Konfig.Res_29 := FALSE;
   BB2_DF.Konfig.Res_30 := FALSE;
   BB2_DF.Konfig.Res_31 := FALSE;
   BB2_DF.MW_EW := 0.0;
   BB2_DF.MW_OG := 100.0;
   BB2_DF.MW_UG := 0.0;
   BB2_DF.GW_HH := 100.0;
   BB2_DF.GW_H := 100.0;
   BB2_DF.GW_L := 0.0;
   BB2_DF.GW_LL := 0.0;
   BB2_DF.GW_Hyst := 1.0;
   BB2_DF.VZ_St := 5;
   BB2_DF.VZ_Ex := 15;
   BB2_DF.MW_Avg := 10;
   Zulauf_Niv.Konfig.Peri := TRUE;
   Zulauf_Niv.Konfig.PW := FALSE;
   Zulauf_Niv.Konfig.Peri_0_20mA := FALSE;
   Zulauf_Niv.Konfig.Peri_4_20mA := TRUE;
   Zulauf_Niv.Konfig.Peri_PT100 := FALSE;
   Zulauf_Niv.Konfig.GW_Delta := FALSE;
   Zulauf_Niv.Konfig.Res_6 := FALSE;
   Zulauf_Niv.Konfig.Res_7 := FALSE;
   Zulauf_Niv.Konfig.Res_8 := FALSE;
   Zulauf_Niv.Konfig.Res_9 := FALSE;
   Zulauf_Niv.Konfig.Res_10 := FALSE;
   Zulauf_Niv.Konfig.Res_11 := FALSE;
   Zulauf_Niv.Konfig.Res_12 := FALSE;
   Zulauf_Niv.Konfig.Res_13 := FALSE;
   Zulauf_Niv.Konfig.Res_14 := FALSE;
   Zulauf_Niv.Konfig.Res_15 := FALSE;
   Zulauf_Niv.Konfig.Res_16 := FALSE;
   Zulauf_Niv.Konfig.Res_17 := FALSE;
   Zulauf_Niv.Konfig.Res_18 := FALSE;
   Zulauf_Niv.Konfig.Res_19 := FALSE;
   Zulauf_Niv.Konfig.Res_20 := FALSE;
   Zulauf_Niv.Konfig.Res_21 := FALSE;
   Zulauf_Niv.Konfig.Res_22 := FALSE;
   Zulauf_Niv.Konfig.Res_23 := FALSE;
   Zulauf_Niv.Konfig.Res_24 := FALSE;
   Zulauf_Niv.Konfig.Res_25 := FALSE;
   Zulauf_Niv.Konfig.Res_26 := FALSE;
   Zulauf_Niv.Konfig.Res_27 := FALSE;
   Zulauf_Niv.Konfig.Res_28 := FALSE;
   Zulauf_Niv.Konfig.Res_29 := FALSE;
   Zulauf_Niv.Konfig.Res_30 := FALSE;
   Zulauf_Niv.Konfig.Res_31 := FALSE;
   Zulauf_Niv.MW_EW := 0.0;
   Zulauf_Niv.MW_OG := 100.0;
   Zulauf_Niv.MW_UG := 0.0;
   Zulauf_Niv.GW_HH := 90.0;
   Zulauf_Niv.GW_H := 60.0;
   Zulauf_Niv.GW_L := 0.0;
   Zulauf_Niv.GW_LL := 0.0;
   Zulauf_Niv.GW_Hyst := 1.0;
   Zulauf_Niv.VZ_St := 5;
   Zulauf_Niv.VZ_Ex := 15;
   Zulauf_Niv.MW_Avg := 10;
   Zulauf_DF.Konfig.Peri := TRUE;
   Zulauf_DF.Konfig.PW := FALSE;
   Zulauf_DF.Konfig.Peri_0_20mA := FALSE;
   Zulauf_DF.Konfig.Peri_4_20mA := TRUE;
   Zulauf_DF.Konfig.Peri_PT100 := FALSE;
   Zulauf_DF.Konfig.GW_Delta := FALSE;
   Zulauf_DF.Konfig.Res_6 := FALSE;
   Zulauf_DF.Konfig.Res_7 := FALSE;
   Zulauf_DF.Konfig.Res_8 := FALSE;
   Zulauf_DF.Konfig.Res_9 := FALSE;
   Zulauf_DF.Konfig.Res_10 := FALSE;
   Zulauf_DF.Konfig.Res_11 := FALSE;
   Zulauf_DF.Konfig.Res_12 := FALSE;
   Zulauf_DF.Konfig.Res_13 := FALSE;
   Zulauf_DF.Konfig.Res_14 := FALSE;
   Zulauf_DF.Konfig.Res_15 := FALSE;
   Zulauf_DF.Konfig.Res_16 := FALSE;
   Zulauf_DF.Konfig.Res_17 := FALSE;
   Zulauf_DF.Konfig.Res_18 := FALSE;
   Zulauf_DF.Konfig.Res_19 := FALSE;
   Zulauf_DF.Konfig.Res_20 := FALSE;
   Zulauf_DF.Konfig.Res_21 := FALSE;
   Zulauf_DF.Konfig.Res_22 := FALSE;
   Zulauf_DF.Konfig.Res_23 := FALSE;
   Zulauf_DF.Konfig.Res_24 := FALSE;
   Zulauf_DF.Konfig.Res_25 := FALSE;
   Zulauf_DF.Konfig.Res_26 := FALSE;
   Zulauf_DF.Konfig.Res_27 := FALSE;
   Zulauf_DF.Konfig.Res_28 := FALSE;
   Zulauf_DF.Konfig.Res_29 := FALSE;
   Zulauf_DF.Konfig.Res_30 := FALSE;
   Zulauf_DF.Konfig.Res_31 := FALSE;
   Zulauf_DF.MW_EW := 0.0;
   Zulauf_DF.MW_OG := 50.0;
   Zulauf_DF.MW_UG := 0.0;
   Zulauf_DF.GW_HH := 40.0;
   Zulauf_DF.GW_H := 40.0;
   Zulauf_DF.GW_L := 0.0;
   Zulauf_DF.GW_LL := 0.0;
   Zulauf_DF.GW_Hyst := 1.0;
   Zulauf_DF.VZ_St := 1800;
   Zulauf_DF.VZ_Ex := 15;
   Zulauf_DF.MW_Avg := 10;
   Verteiler_pH.Konfig.Peri := TRUE;
   Verteiler_pH.Konfig.PW := FALSE;
   Verteiler_pH.Konfig.Peri_0_20mA := FALSE;
   Verteiler_pH.Konfig.Peri_4_20mA := TRUE;
   Verteiler_pH.Konfig.Peri_PT100 := FALSE;
   Verteiler_pH.Konfig.GW_Delta := FALSE;
   Verteiler_pH.Konfig.Res_6 := FALSE;
   Verteiler_pH.Konfig.Res_7 := FALSE;
   Verteiler_pH.Konfig.Res_8 := FALSE;
   Verteiler_pH.Konfig.Res_9 := FALSE;
   Verteiler_pH.Konfig.Res_10 := FALSE;
   Verteiler_pH.Konfig.Res_11 := FALSE;
   Verteiler_pH.Konfig.Res_12 := FALSE;
   Verteiler_pH.Konfig.Res_13 := FALSE;
   Verteiler_pH.Konfig.Res_14 := FALSE;
   Verteiler_pH.Konfig.Res_15 := FALSE;
   Verteiler_pH.Konfig.Res_16 := FALSE;
   Verteiler_pH.Konfig.Res_17 := FALSE;
   Verteiler_pH.Konfig.Res_18 := FALSE;
   Verteiler_pH.Konfig.Res_19 := FALSE;
   Verteiler_pH.Konfig.Res_20 := FALSE;
   Verteiler_pH.Konfig.Res_21 := FALSE;
   Verteiler_pH.Konfig.Res_22 := FALSE;
   Verteiler_pH.Konfig.Res_23 := FALSE;
   Verteiler_pH.Konfig.Res_24 := FALSE;
   Verteiler_pH.Konfig.Res_25 := FALSE;
   Verteiler_pH.Konfig.Res_26 := FALSE;
   Verteiler_pH.Konfig.Res_27 := FALSE;
   Verteiler_pH.Konfig.Res_28 := FALSE;
   Verteiler_pH.Konfig.Res_29 := FALSE;
   Verteiler_pH.Konfig.Res_30 := FALSE;
   Verteiler_pH.Konfig.Res_31 := FALSE;
   Verteiler_pH.MW_EW := 0.0;
   Verteiler_pH.MW_OG := 12.0;
   Verteiler_pH.MW_UG := 2.0;
   Verteiler_pH.GW_HH := 12.0;
   Verteiler_pH.GW_H := 12.0;
   Verteiler_pH.GW_L := 2.0;
   Verteiler_pH.GW_LL := 2.0;
   Verteiler_pH.GW_Hyst := 1.0;
   Verteiler_pH.VZ_St := 5;
   Verteiler_pH.VZ_Ex := 15;
   Verteiler_pH.MW_Avg := 10;
   Verteiler_O2.Konfig.Peri := TRUE;
   Verteiler_O2.Konfig.PW := FALSE;
   Verteiler_O2.Konfig.Peri_0_20mA := FALSE;
   Verteiler_O2.Konfig.Peri_4_20mA := TRUE;
   Verteiler_O2.Konfig.Peri_PT100 := FALSE;
   Verteiler_O2.Konfig.GW_Delta := FALSE;
   Verteiler_O2.Konfig.Res_6 := FALSE;
   Verteiler_O2.Konfig.Res_7 := FALSE;
   Verteiler_O2.Konfig.Res_8 := FALSE;
   Verteiler_O2.Konfig.Res_9 := FALSE;
   Verteiler_O2.Konfig.Res_10 := FALSE;
   Verteiler_O2.Konfig.Res_11 := FALSE;
   Verteiler_O2.Konfig.Res_12 := FALSE;
   Verteiler_O2.Konfig.Res_13 := FALSE;
   Verteiler_O2.Konfig.Res_14 := FALSE;
   Verteiler_O2.Konfig.Res_15 := FALSE;
   Verteiler_O2.Konfig.Res_16 := FALSE;
   Verteiler_O2.Konfig.Res_17 := FALSE;
   Verteiler_O2.Konfig.Res_18 := FALSE;
   Verteiler_O2.Konfig.Res_19 := FALSE;
   Verteiler_O2.Konfig.Res_20 := FALSE;
   Verteiler_O2.Konfig.Res_21 := FALSE;
   Verteiler_O2.Konfig.Res_22 := FALSE;
   Verteiler_O2.Konfig.Res_23 := FALSE;
   Verteiler_O2.Konfig.Res_24 := FALSE;
   Verteiler_O2.Konfig.Res_25 := FALSE;
   Verteiler_O2.Konfig.Res_26 := FALSE;
   Verteiler_O2.Konfig.Res_27 := FALSE;
   Verteiler_O2.Konfig.Res_28 := FALSE;
   Verteiler_O2.Konfig.Res_29 := FALSE;
   Verteiler_O2.Konfig.Res_30 := FALSE;
   Verteiler_O2.Konfig.Res_31 := FALSE;
   Verteiler_O2.MW_EW := 0.0;
   Verteiler_O2.MW_OG := 10.0;
   Verteiler_O2.MW_UG := 0.0;
   Verteiler_O2.GW_HH := 10.0;
   Verteiler_O2.GW_H := 10.0;
   Verteiler_O2.GW_L := 0.0;
   Verteiler_O2.GW_LL := 0.0;
   Verteiler_O2.GW_Hyst := 1.0;
   Verteiler_O2.VZ_St := 5;
   Verteiler_O2.VZ_Ex := 15;
   Verteiler_O2.MW_Avg := 20;
   Verteiler_Temp.Konfig.Peri := TRUE;
   Verteiler_Temp.Konfig.PW := FALSE;
   Verteiler_Temp.Konfig.Peri_0_20mA := FALSE;
   Verteiler_Temp.Konfig.Peri_4_20mA := TRUE;
   Verteiler_Temp.Konfig.Peri_PT100 := FALSE;
   Verteiler_Temp.Konfig.GW_Delta := FALSE;
   Verteiler_Temp.Konfig.Res_6 := FALSE;
   Verteiler_Temp.Konfig.Res_7 := FALSE;
   Verteiler_Temp.Konfig.Res_8 := FALSE;
   Verteiler_Temp.Konfig.Res_9 := FALSE;
   Verteiler_Temp.Konfig.Res_10 := FALSE;
   Verteiler_Temp.Konfig.Res_11 := FALSE;
   Verteiler_Temp.Konfig.Res_12 := FALSE;
   Verteiler_Temp.Konfig.Res_13 := FALSE;
   Verteiler_Temp.Konfig.Res_14 := FALSE;
   Verteiler_Temp.Konfig.Res_15 := FALSE;
   Verteiler_Temp.Konfig.Res_16 := FALSE;
   Verteiler_Temp.Konfig.Res_17 := FALSE;
   Verteiler_Temp.Konfig.Res_18 := FALSE;
   Verteiler_Temp.Konfig.Res_19 := FALSE;
   Verteiler_Temp.Konfig.Res_20 := FALSE;
   Verteiler_Temp.Konfig.Res_21 := FALSE;
   Verteiler_Temp.Konfig.Res_22 := FALSE;
   Verteiler_Temp.Konfig.Res_23 := FALSE;
   Verteiler_Temp.Konfig.Res_24 := FALSE;
   Verteiler_Temp.Konfig.Res_25 := FALSE;
   Verteiler_Temp.Konfig.Res_26 := FALSE;
   Verteiler_Temp.Konfig.Res_27 := FALSE;
   Verteiler_Temp.Konfig.Res_28 := FALSE;
   Verteiler_Temp.Konfig.Res_29 := FALSE;
   Verteiler_Temp.Konfig.Res_30 := FALSE;
   Verteiler_Temp.Konfig.Res_31 := FALSE;
   Verteiler_Temp.MW_EW := 0.0;
   Verteiler_Temp.MW_OG := 50.0;
   Verteiler_Temp.MW_UG := 0.0;
   Verteiler_Temp.GW_HH := 50.0;
   Verteiler_Temp.GW_H := 50.0;
   Verteiler_Temp.GW_L := 0.0;
   Verteiler_Temp.GW_LL := 0.0;
   Verteiler_Temp.GW_Hyst := 1.0;
   Verteiler_Temp.VZ_St := 5;
   Verteiler_Temp.VZ_Ex := 15;
   Verteiler_Temp.MW_Avg := 30;
   BB_UeSS_DF.Konfig.Peri := TRUE;
   BB_UeSS_DF.Konfig.PW := FALSE;
   BB_UeSS_DF.Konfig.Peri_0_20mA := FALSE;
   BB_UeSS_DF.Konfig.Peri_4_20mA := TRUE;
   BB_UeSS_DF.Konfig.Peri_PT100 := FALSE;
   BB_UeSS_DF.Konfig.GW_Delta := FALSE;
   BB_UeSS_DF.Konfig.Res_6 := FALSE;
   BB_UeSS_DF.Konfig.Res_7 := FALSE;
   BB_UeSS_DF.Konfig.Res_8 := FALSE;
   BB_UeSS_DF.Konfig.Res_9 := FALSE;
   BB_UeSS_DF.Konfig.Res_10 := FALSE;
   BB_UeSS_DF.Konfig.Res_11 := FALSE;
   BB_UeSS_DF.Konfig.Res_12 := FALSE;
   BB_UeSS_DF.Konfig.Res_13 := FALSE;
   BB_UeSS_DF.Konfig.Res_14 := FALSE;
   BB_UeSS_DF.Konfig.Res_15 := FALSE;
   BB_UeSS_DF.Konfig.Res_16 := FALSE;
   BB_UeSS_DF.Konfig.Res_17 := FALSE;
   BB_UeSS_DF.Konfig.Res_18 := FALSE;
   BB_UeSS_DF.Konfig.Res_19 := FALSE;
   BB_UeSS_DF.Konfig.Res_20 := FALSE;
   BB_UeSS_DF.Konfig.Res_21 := FALSE;
   BB_UeSS_DF.Konfig.Res_22 := FALSE;
   BB_UeSS_DF.Konfig.Res_23 := FALSE;
   BB_UeSS_DF.Konfig.Res_24 := FALSE;
   BB_UeSS_DF.Konfig.Res_25 := FALSE;
   BB_UeSS_DF.Konfig.Res_26 := FALSE;
   BB_UeSS_DF.Konfig.Res_27 := FALSE;
   BB_UeSS_DF.Konfig.Res_28 := FALSE;
   BB_UeSS_DF.Konfig.Res_29 := FALSE;
   BB_UeSS_DF.Konfig.Res_30 := FALSE;
   BB_UeSS_DF.Konfig.Res_31 := FALSE;
   BB_UeSS_DF.MW_EW := 0.0;
   BB_UeSS_DF.MW_OG := 20.0;
   BB_UeSS_DF.MW_UG := 0.0;
   BB_UeSS_DF.GW_HH := 10.0;
   BB_UeSS_DF.GW_H := 10.0;
   BB_UeSS_DF.GW_L := 0.5;
   BB_UeSS_DF.GW_LL := 0.5;
   BB_UeSS_DF.GW_Hyst := 1.0;
   BB_UeSS_DF.VZ_St := 5;
   BB_UeSS_DF.VZ_Ex := 15;
   BB_UeSS_DF.MW_Avg := 10;
   Ablauf_DF.Konfig.Peri := TRUE;
   Ablauf_DF.Konfig.PW := FALSE;
   Ablauf_DF.Konfig.Peri_0_20mA := FALSE;
   Ablauf_DF.Konfig.Peri_4_20mA := TRUE;
   Ablauf_DF.Konfig.Peri_PT100 := FALSE;
   Ablauf_DF.Konfig.GW_Delta := FALSE;
   Ablauf_DF.Konfig.Res_6 := FALSE;
   Ablauf_DF.Konfig.Res_7 := FALSE;
   Ablauf_DF.Konfig.Res_8 := FALSE;
   Ablauf_DF.Konfig.Res_9 := FALSE;
   Ablauf_DF.Konfig.Res_10 := FALSE;
   Ablauf_DF.Konfig.Res_11 := FALSE;
   Ablauf_DF.Konfig.Res_12 := FALSE;
   Ablauf_DF.Konfig.Res_13 := FALSE;
   Ablauf_DF.Konfig.Res_14 := FALSE;
   Ablauf_DF.Konfig.Res_15 := FALSE;
   Ablauf_DF.Konfig.Res_16 := FALSE;
   Ablauf_DF.Konfig.Res_17 := FALSE;
   Ablauf_DF.Konfig.Res_18 := FALSE;
   Ablauf_DF.Konfig.Res_19 := FALSE;
   Ablauf_DF.Konfig.Res_20 := FALSE;
   Ablauf_DF.Konfig.Res_21 := FALSE;
   Ablauf_DF.Konfig.Res_22 := FALSE;
   Ablauf_DF.Konfig.Res_23 := FALSE;
   Ablauf_DF.Konfig.Res_24 := FALSE;
   Ablauf_DF.Konfig.Res_25 := FALSE;
   Ablauf_DF.Konfig.Res_26 := FALSE;
   Ablauf_DF.Konfig.Res_27 := FALSE;
   Ablauf_DF.Konfig.Res_28 := FALSE;
   Ablauf_DF.Konfig.Res_29 := FALSE;
   Ablauf_DF.Konfig.Res_30 := FALSE;
   Ablauf_DF.Konfig.Res_31 := FALSE;
   Ablauf_DF.MW_EW := 0.0;
   Ablauf_DF.MW_OG := 30.0;
   Ablauf_DF.MW_UG := 0.0;
   Ablauf_DF.GW_HH := 30.0;
   Ablauf_DF.GW_H := 30.0;
   Ablauf_DF.GW_L := 0.0;
   Ablauf_DF.GW_LL := 0.0;
   Ablauf_DF.GW_Hyst := 1.0;
   Ablauf_DF.VZ_St := 5;
   Ablauf_DF.VZ_Ex := 15;
   Ablauf_DF.MW_Avg := 10;
   Ablauf_pH.Konfig.Peri := TRUE;
   Ablauf_pH.Konfig.PW := FALSE;
   Ablauf_pH.Konfig.Peri_0_20mA := FALSE;
   Ablauf_pH.Konfig.Peri_4_20mA := TRUE;
   Ablauf_pH.Konfig.Peri_PT100 := FALSE;
   Ablauf_pH.Konfig.GW_Delta := FALSE;
   Ablauf_pH.Konfig.Res_6 := FALSE;
   Ablauf_pH.Konfig.Res_7 := FALSE;
   Ablauf_pH.Konfig.Res_8 := FALSE;
   Ablauf_pH.Konfig.Res_9 := FALSE;
   Ablauf_pH.Konfig.Res_10 := FALSE;
   Ablauf_pH.Konfig.Res_11 := FALSE;
   Ablauf_pH.Konfig.Res_12 := FALSE;
   Ablauf_pH.Konfig.Res_13 := FALSE;
   Ablauf_pH.Konfig.Res_14 := FALSE;
   Ablauf_pH.Konfig.Res_15 := FALSE;
   Ablauf_pH.Konfig.Res_16 := FALSE;
   Ablauf_pH.Konfig.Res_17 := FALSE;
   Ablauf_pH.Konfig.Res_18 := FALSE;
   Ablauf_pH.Konfig.Res_19 := FALSE;
   Ablauf_pH.Konfig.Res_20 := FALSE;
   Ablauf_pH.Konfig.Res_21 := FALSE;
   Ablauf_pH.Konfig.Res_22 := FALSE;
   Ablauf_pH.Konfig.Res_23 := FALSE;
   Ablauf_pH.Konfig.Res_24 := FALSE;
   Ablauf_pH.Konfig.Res_25 := FALSE;
   Ablauf_pH.Konfig.Res_26 := FALSE;
   Ablauf_pH.Konfig.Res_27 := FALSE;
   Ablauf_pH.Konfig.Res_28 := FALSE;
   Ablauf_pH.Konfig.Res_29 := FALSE;
   Ablauf_pH.Konfig.Res_30 := FALSE;
   Ablauf_pH.Konfig.Res_31 := FALSE;
   Ablauf_pH.MW_EW := 0.0;
   Ablauf_pH.MW_OG := 14.0;
   Ablauf_pH.MW_UG := 0.0;
   Ablauf_pH.GW_HH := 14.0;
   Ablauf_pH.GW_H := 14.0;
   Ablauf_pH.GW_L := 0.0;
   Ablauf_pH.GW_LL := 0.0;
   Ablauf_pH.GW_Hyst := 1.0;
   Ablauf_pH.VZ_St := 5;
   Ablauf_pH.VZ_Ex := 15;
   Ablauf_pH.MW_Avg := 10;
   Ablauf_O2.Konfig.Peri := TRUE;
   Ablauf_O2.Konfig.PW := FALSE;
   Ablauf_O2.Konfig.Peri_0_20mA := FALSE;
   Ablauf_O2.Konfig.Peri_4_20mA := TRUE;
   Ablauf_O2.Konfig.Peri_PT100 := FALSE;
   Ablauf_O2.Konfig.GW_Delta := FALSE;
   Ablauf_O2.Konfig.Res_6 := FALSE;
   Ablauf_O2.Konfig.Res_7 := FALSE;
   Ablauf_O2.Konfig.Res_8 := FALSE;
   Ablauf_O2.Konfig.Res_9 := FALSE;
   Ablauf_O2.Konfig.Res_10 := FALSE;
   Ablauf_O2.Konfig.Res_11 := FALSE;
   Ablauf_O2.Konfig.Res_12 := FALSE;
   Ablauf_O2.Konfig.Res_13 := FALSE;
   Ablauf_O2.Konfig.Res_14 := FALSE;
   Ablauf_O2.Konfig.Res_15 := FALSE;
   Ablauf_O2.Konfig.Res_16 := FALSE;
   Ablauf_O2.Konfig.Res_17 := FALSE;
   Ablauf_O2.Konfig.Res_18 := FALSE;
   Ablauf_O2.Konfig.Res_19 := FALSE;
   Ablauf_O2.Konfig.Res_20 := FALSE;
   Ablauf_O2.Konfig.Res_21 := FALSE;
   Ablauf_O2.Konfig.Res_22 := FALSE;
   Ablauf_O2.Konfig.Res_23 := FALSE;
   Ablauf_O2.Konfig.Res_24 := FALSE;
   Ablauf_O2.Konfig.Res_25 := FALSE;
   Ablauf_O2.Konfig.Res_26 := FALSE;
   Ablauf_O2.Konfig.Res_27 := FALSE;
   Ablauf_O2.Konfig.Res_28 := FALSE;
   Ablauf_O2.Konfig.Res_29 := FALSE;
   Ablauf_O2.Konfig.Res_30 := FALSE;
   Ablauf_O2.Konfig.Res_31 := FALSE;
   Ablauf_O2.MW_EW := 0.0;
   Ablauf_O2.MW_OG := 10.0;
   Ablauf_O2.MW_UG := 0.0;
   Ablauf_O2.GW_HH := 10.0;
   Ablauf_O2.GW_H := 10.0;
   Ablauf_O2.GW_L := 0.0;
   Ablauf_O2.GW_LL := 0.0;
   Ablauf_O2.GW_Hyst := 1.0;
   Ablauf_O2.VZ_St := 5;
   Ablauf_O2.VZ_Ex := 15;
   Ablauf_O2.MW_Avg := 10;
   Ablauf_Temp.Konfig.Peri := TRUE;
   Ablauf_Temp.Konfig.PW := FALSE;
   Ablauf_Temp.Konfig.Peri_0_20mA := FALSE;
   Ablauf_Temp.Konfig.Peri_4_20mA := TRUE;
   Ablauf_Temp.Konfig.Peri_PT100 := FALSE;
   Ablauf_Temp.Konfig.GW_Delta := FALSE;
   Ablauf_Temp.Konfig.Res_6 := FALSE;
   Ablauf_Temp.Konfig.Res_7 := FALSE;
   Ablauf_Temp.Konfig.Res_8 := FALSE;
   Ablauf_Temp.Konfig.Res_9 := FALSE;
   Ablauf_Temp.Konfig.Res_10 := FALSE;
   Ablauf_Temp.Konfig.Res_11 := FALSE;
   Ablauf_Temp.Konfig.Res_12 := FALSE;
   Ablauf_Temp.Konfig.Res_13 := FALSE;
   Ablauf_Temp.Konfig.Res_14 := FALSE;
   Ablauf_Temp.Konfig.Res_15 := FALSE;
   Ablauf_Temp.Konfig.Res_16 := FALSE;
   Ablauf_Temp.Konfig.Res_17 := FALSE;
   Ablauf_Temp.Konfig.Res_18 := FALSE;
   Ablauf_Temp.Konfig.Res_19 := FALSE;
   Ablauf_Temp.Konfig.Res_20 := FALSE;
   Ablauf_Temp.Konfig.Res_21 := FALSE;
   Ablauf_Temp.Konfig.Res_22 := FALSE;
   Ablauf_Temp.Konfig.Res_23 := FALSE;
   Ablauf_Temp.Konfig.Res_24 := FALSE;
   Ablauf_Temp.Konfig.Res_25 := FALSE;
   Ablauf_Temp.Konfig.Res_26 := FALSE;
   Ablauf_Temp.Konfig.Res_27 := FALSE;
   Ablauf_Temp.Konfig.Res_28 := FALSE;
   Ablauf_Temp.Konfig.Res_29 := FALSE;
   Ablauf_Temp.Konfig.Res_30 := FALSE;
   Ablauf_Temp.Konfig.Res_31 := FALSE;
   Ablauf_Temp.MW_EW := 0.0;
   Ablauf_Temp.MW_OG := 50.0;
   Ablauf_Temp.MW_UG := 0.0;
   Ablauf_Temp.GW_HH := 40.0;
   Ablauf_Temp.GW_H := 40.0;
   Ablauf_Temp.GW_L := 0.0;
   Ablauf_Temp.GW_LL := 0.0;
   Ablauf_Temp.GW_Hyst := 1.0;
   Ablauf_Temp.VZ_St := 5;
   Ablauf_Temp.VZ_Ex := 15;
   Ablauf_Temp.MW_Avg := 10;
   Schlamm_ED_Niv.Konfig.Peri := TRUE;
   Schlamm_ED_Niv.Konfig.PW := FALSE;
   Schlamm_ED_Niv.Konfig.Peri_0_20mA := FALSE;
   Schlamm_ED_Niv.Konfig.Peri_4_20mA := TRUE;
   Schlamm_ED_Niv.Konfig.Peri_PT100 := FALSE;
   Schlamm_ED_Niv.Konfig.GW_Delta := FALSE;
   Schlamm_ED_Niv.Konfig.Res_6 := FALSE;
   Schlamm_ED_Niv.Konfig.Res_7 := FALSE;
   Schlamm_ED_Niv.Konfig.Res_8 := FALSE;
   Schlamm_ED_Niv.Konfig.Res_9 := FALSE;
   Schlamm_ED_Niv.Konfig.Res_10 := FALSE;
   Schlamm_ED_Niv.Konfig.Res_11 := FALSE;
   Schlamm_ED_Niv.Konfig.Res_12 := FALSE;
   Schlamm_ED_Niv.Konfig.Res_13 := FALSE;
   Schlamm_ED_Niv.Konfig.Res_14 := FALSE;
   Schlamm_ED_Niv.Konfig.Res_15 := FALSE;
   Schlamm_ED_Niv.Konfig.Res_16 := FALSE;
   Schlamm_ED_Niv.Konfig.Res_17 := FALSE;
   Schlamm_ED_Niv.Konfig.Res_18 := FALSE;
   Schlamm_ED_Niv.Konfig.Res_19 := FALSE;
   Schlamm_ED_Niv.Konfig.Res_20 := FALSE;
   Schlamm_ED_Niv.Konfig.Res_21 := FALSE;
   Schlamm_ED_Niv.Konfig.Res_22 := FALSE;
   Schlamm_ED_Niv.Konfig.Res_23 := FALSE;
   Schlamm_ED_Niv.Konfig.Res_24 := FALSE;
   Schlamm_ED_Niv.Konfig.Res_25 := FALSE;
   Schlamm_ED_Niv.Konfig.Res_26 := FALSE;
   Schlamm_ED_Niv.Konfig.Res_27 := FALSE;
   Schlamm_ED_Niv.Konfig.Res_28 := FALSE;
   Schlamm_ED_Niv.Konfig.Res_29 := FALSE;
   Schlamm_ED_Niv.Konfig.Res_30 := FALSE;
   Schlamm_ED_Niv.Konfig.Res_31 := FALSE;
   Schlamm_ED_Niv.MW_EW := 0.0;
   Schlamm_ED_Niv.MW_OG := 100.0;
   Schlamm_ED_Niv.MW_UG := 0.0;
   Schlamm_ED_Niv.GW_HH := 100.0;
   Schlamm_ED_Niv.GW_H := 100.0;
   Schlamm_ED_Niv.GW_L := 0.0;
   Schlamm_ED_Niv.GW_LL := 0.0;
   Schlamm_ED_Niv.GW_Hyst := 1.0;
   Schlamm_ED_Niv.VZ_St := 5;
   Schlamm_ED_Niv.VZ_Ex := 15;
   Schlamm_ED_Niv.MW_Avg := 30;
   Schlamm_Besch_Niv.Konfig.Peri := TRUE;
   Schlamm_Besch_Niv.Konfig.PW := FALSE;
   Schlamm_Besch_Niv.Konfig.Peri_0_20mA := FALSE;
   Schlamm_Besch_Niv.Konfig.Peri_4_20mA := TRUE;
   Schlamm_Besch_Niv.Konfig.Peri_PT100 := FALSE;
   Schlamm_Besch_Niv.Konfig.GW_Delta := FALSE;
   Schlamm_Besch_Niv.Konfig.Res_6 := FALSE;
   Schlamm_Besch_Niv.Konfig.Res_7 := FALSE;
   Schlamm_Besch_Niv.Konfig.Res_8 := FALSE;
   Schlamm_Besch_Niv.Konfig.Res_9 := FALSE;
   Schlamm_Besch_Niv.Konfig.Res_10 := FALSE;
   Schlamm_Besch_Niv.Konfig.Res_11 := FALSE;
   Schlamm_Besch_Niv.Konfig.Res_12 := FALSE;
   Schlamm_Besch_Niv.Konfig.Res_13 := FALSE;
   Schlamm_Besch_Niv.Konfig.Res_14 := FALSE;
   Schlamm_Besch_Niv.Konfig.Res_15 := FALSE;
   Schlamm_Besch_Niv.Konfig.Res_16 := FALSE;
   Schlamm_Besch_Niv.Konfig.Res_17 := FALSE;
   Schlamm_Besch_Niv.Konfig.Res_18 := FALSE;
   Schlamm_Besch_Niv.Konfig.Res_19 := FALSE;
   Schlamm_Besch_Niv.Konfig.Res_20 := FALSE;
   Schlamm_Besch_Niv.Konfig.Res_21 := FALSE;
   Schlamm_Besch_Niv.Konfig.Res_22 := FALSE;
   Schlamm_Besch_Niv.Konfig.Res_23 := FALSE;
   Schlamm_Besch_Niv.Konfig.Res_24 := FALSE;
   Schlamm_Besch_Niv.Konfig.Res_25 := FALSE;
   Schlamm_Besch_Niv.Konfig.Res_26 := FALSE;
   Schlamm_Besch_Niv.Konfig.Res_27 := FALSE;
   Schlamm_Besch_Niv.Konfig.Res_28 := FALSE;
   Schlamm_Besch_Niv.Konfig.Res_29 := FALSE;
   Schlamm_Besch_Niv.Konfig.Res_30 := FALSE;
   Schlamm_Besch_Niv.Konfig.Res_31 := FALSE;
   Schlamm_Besch_Niv.MW_EW := 0.0;
   Schlamm_Besch_Niv.MW_OG := 100.0;
   Schlamm_Besch_Niv.MW_UG := 0.0;
   Schlamm_Besch_Niv.GW_HH := 100.0;
   Schlamm_Besch_Niv.GW_H := 100.0;
   Schlamm_Besch_Niv.GW_L := 0.0;
   Schlamm_Besch_Niv.GW_LL := 0.0;
   Schlamm_Besch_Niv.GW_Hyst := 1.0;
   Schlamm_Besch_Niv.VZ_St := 5;
   Schlamm_Besch_Niv.VZ_Ex := 15;
   Schlamm_Besch_Niv.MW_Avg := 30;
   Schlamm_Besch_DF.Konfig.Peri := TRUE;
   Schlamm_Besch_DF.Konfig.PW := FALSE;
   Schlamm_Besch_DF.Konfig.Peri_0_20mA := FALSE;
   Schlamm_Besch_DF.Konfig.Peri_4_20mA := TRUE;
   Schlamm_Besch_DF.Konfig.Peri_PT100 := FALSE;
   Schlamm_Besch_DF.Konfig.GW_Delta := FALSE;
   Schlamm_Besch_DF.Konfig.Res_6 := FALSE;
   Schlamm_Besch_DF.Konfig.Res_7 := FALSE;
   Schlamm_Besch_DF.Konfig.Res_8 := FALSE;
   Schlamm_Besch_DF.Konfig.Res_9 := FALSE;
   Schlamm_Besch_DF.Konfig.Res_10 := FALSE;
   Schlamm_Besch_DF.Konfig.Res_11 := FALSE;
   Schlamm_Besch_DF.Konfig.Res_12 := FALSE;
   Schlamm_Besch_DF.Konfig.Res_13 := FALSE;
   Schlamm_Besch_DF.Konfig.Res_14 := FALSE;
   Schlamm_Besch_DF.Konfig.Res_15 := FALSE;
   Schlamm_Besch_DF.Konfig.Res_16 := FALSE;
   Schlamm_Besch_DF.Konfig.Res_17 := FALSE;
   Schlamm_Besch_DF.Konfig.Res_18 := FALSE;
   Schlamm_Besch_DF.Konfig.Res_19 := FALSE;
   Schlamm_Besch_DF.Konfig.Res_20 := FALSE;
   Schlamm_Besch_DF.Konfig.Res_21 := FALSE;
   Schlamm_Besch_DF.Konfig.Res_22 := FALSE;
   Schlamm_Besch_DF.Konfig.Res_23 := FALSE;
   Schlamm_Besch_DF.Konfig.Res_24 := FALSE;
   Schlamm_Besch_DF.Konfig.Res_25 := FALSE;
   Schlamm_Besch_DF.Konfig.Res_26 := FALSE;
   Schlamm_Besch_DF.Konfig.Res_27 := FALSE;
   Schlamm_Besch_DF.Konfig.Res_28 := FALSE;
   Schlamm_Besch_DF.Konfig.Res_29 := FALSE;
   Schlamm_Besch_DF.Konfig.Res_30 := FALSE;
   Schlamm_Besch_DF.Konfig.Res_31 := FALSE;
   Schlamm_Besch_DF.MW_EW := 0.0;
   Schlamm_Besch_DF.MW_OG := 20.0;
   Schlamm_Besch_DF.MW_UG := 0.0;
   Schlamm_Besch_DF.GW_HH := 25.0;
   Schlamm_Besch_DF.GW_H := 20.0;
   Schlamm_Besch_DF.GW_L := 0.0;
   Schlamm_Besch_DF.GW_LL := 0.0;
   Schlamm_Besch_DF.GW_Hyst := 1.0;
   Schlamm_Besch_DF.VZ_St := 5;
   Schlamm_Besch_DF.VZ_Ex := 15;
   Schlamm_Besch_DF.MW_Avg := 10;
   Truebwasser_Niv.Konfig.Peri := TRUE;
   Truebwasser_Niv.Konfig.PW := FALSE;
   Truebwasser_Niv.Konfig.Peri_0_20mA := FALSE;
   Truebwasser_Niv.Konfig.Peri_4_20mA := TRUE;
   Truebwasser_Niv.Konfig.Peri_PT100 := FALSE;
   Truebwasser_Niv.Konfig.GW_Delta := FALSE;
   Truebwasser_Niv.Konfig.Res_6 := FALSE;
   Truebwasser_Niv.Konfig.Res_7 := FALSE;
   Truebwasser_Niv.Konfig.Res_8 := FALSE;
   Truebwasser_Niv.Konfig.Res_9 := FALSE;
   Truebwasser_Niv.Konfig.Res_10 := FALSE;
   Truebwasser_Niv.Konfig.Res_11 := FALSE;
   Truebwasser_Niv.Konfig.Res_12 := FALSE;
   Truebwasser_Niv.Konfig.Res_13 := FALSE;
   Truebwasser_Niv.Konfig.Res_14 := FALSE;
   Truebwasser_Niv.Konfig.Res_15 := FALSE;
   Truebwasser_Niv.Konfig.Res_16 := FALSE;
   Truebwasser_Niv.Konfig.Res_17 := FALSE;
   Truebwasser_Niv.Konfig.Res_18 := FALSE;
   Truebwasser_Niv.Konfig.Res_19 := FALSE;
   Truebwasser_Niv.Konfig.Res_20 := FALSE;
   Truebwasser_Niv.Konfig.Res_21 := FALSE;
   Truebwasser_Niv.Konfig.Res_22 := FALSE;
   Truebwasser_Niv.Konfig.Res_23 := FALSE;
   Truebwasser_Niv.Konfig.Res_24 := FALSE;
   Truebwasser_Niv.Konfig.Res_25 := FALSE;
   Truebwasser_Niv.Konfig.Res_26 := FALSE;
   Truebwasser_Niv.Konfig.Res_27 := FALSE;
   Truebwasser_Niv.Konfig.Res_28 := FALSE;
   Truebwasser_Niv.Konfig.Res_29 := FALSE;
   Truebwasser_Niv.Konfig.Res_30 := FALSE;
   Truebwasser_Niv.Konfig.Res_31 := FALSE;
   Truebwasser_Niv.MW_EW := 0.0;
   Truebwasser_Niv.MW_OG := 100.0;
   Truebwasser_Niv.MW_UG := 0.0;
   Truebwasser_Niv.GW_HH := 100.0;
   Truebwasser_Niv.GW_H := 100.0;
   Truebwasser_Niv.GW_L := 0.0;
   Truebwasser_Niv.GW_LL := 0.0;
   Truebwasser_Niv.GW_Hyst := 1.0;
   Truebwasser_Niv.VZ_St := 5;
   Truebwasser_Niv.VZ_Ex := 15;
   Truebwasser_Niv.MW_Avg := 10;
   Truebwasser_DF.Konfig.Peri := TRUE;
   Truebwasser_DF.Konfig.PW := FALSE;
   Truebwasser_DF.Konfig.Peri_0_20mA := FALSE;
   Truebwasser_DF.Konfig.Peri_4_20mA := TRUE;
   Truebwasser_DF.Konfig.Peri_PT100 := FALSE;
   Truebwasser_DF.Konfig.GW_Delta := FALSE;
   Truebwasser_DF.Konfig.Res_6 := FALSE;
   Truebwasser_DF.Konfig.Res_7 := FALSE;
   Truebwasser_DF.Konfig.Res_8 := FALSE;
   Truebwasser_DF.Konfig.Res_9 := FALSE;
   Truebwasser_DF.Konfig.Res_10 := FALSE;
   Truebwasser_DF.Konfig.Res_11 := FALSE;
   Truebwasser_DF.Konfig.Res_12 := FALSE;
   Truebwasser_DF.Konfig.Res_13 := FALSE;
   Truebwasser_DF.Konfig.Res_14 := FALSE;
   Truebwasser_DF.Konfig.Res_15 := FALSE;
   Truebwasser_DF.Konfig.Res_16 := FALSE;
   Truebwasser_DF.Konfig.Res_17 := FALSE;
   Truebwasser_DF.Konfig.Res_18 := FALSE;
   Truebwasser_DF.Konfig.Res_19 := FALSE;
   Truebwasser_DF.Konfig.Res_20 := FALSE;
   Truebwasser_DF.Konfig.Res_21 := FALSE;
   Truebwasser_DF.Konfig.Res_22 := FALSE;
   Truebwasser_DF.Konfig.Res_23 := FALSE;
   Truebwasser_DF.Konfig.Res_24 := FALSE;
   Truebwasser_DF.Konfig.Res_25 := FALSE;
   Truebwasser_DF.Konfig.Res_26 := FALSE;
   Truebwasser_DF.Konfig.Res_27 := FALSE;
   Truebwasser_DF.Konfig.Res_28 := FALSE;
   Truebwasser_DF.Konfig.Res_29 := FALSE;
   Truebwasser_DF.Konfig.Res_30 := FALSE;
   Truebwasser_DF.Konfig.Res_31 := FALSE;
   Truebwasser_DF.MW_EW := 0.0;
   Truebwasser_DF.MW_OG := 25.0;
   Truebwasser_DF.MW_UG := 0.0;
   Truebwasser_DF.GW_HH := 20.0;
   Truebwasser_DF.GW_H := 20.0;
   Truebwasser_DF.GW_L := 0.0;
   Truebwasser_DF.GW_LL := 0.0;
   Truebwasser_DF.GW_Hyst := 1.0;
   Truebwasser_DF.VZ_St := 5;
   Truebwasser_DF.VZ_Ex := 15;
   Truebwasser_DF.MW_Avg := 10;
   Zulauf_SF_Niv.Konfig.Peri := TRUE;
   Zulauf_SF_Niv.Konfig.PW := FALSE;
   Zulauf_SF_Niv.Konfig.Peri_0_20mA := FALSE;
   Zulauf_SF_Niv.Konfig.Peri_4_20mA := TRUE;
   Zulauf_SF_Niv.Konfig.Peri_PT100 := FALSE;
   Zulauf_SF_Niv.Konfig.GW_Delta := FALSE;
   Zulauf_SF_Niv.Konfig.Res_6 := FALSE;
   Zulauf_SF_Niv.Konfig.Res_7 := FALSE;
   Zulauf_SF_Niv.Konfig.Res_8 := FALSE;
   Zulauf_SF_Niv.Konfig.Res_9 := FALSE;
   Zulauf_SF_Niv.Konfig.Res_10 := FALSE;
   Zulauf_SF_Niv.Konfig.Res_11 := FALSE;
   Zulauf_SF_Niv.Konfig.Res_12 := FALSE;
   Zulauf_SF_Niv.Konfig.Res_13 := FALSE;
   Zulauf_SF_Niv.Konfig.Res_14 := FALSE;
   Zulauf_SF_Niv.Konfig.Res_15 := FALSE;
   Zulauf_SF_Niv.Konfig.Res_16 := FALSE;
   Zulauf_SF_Niv.Konfig.Res_17 := FALSE;
   Zulauf_SF_Niv.Konfig.Res_18 := FALSE;
   Zulauf_SF_Niv.Konfig.Res_19 := FALSE;
   Zulauf_SF_Niv.Konfig.Res_20 := FALSE;
   Zulauf_SF_Niv.Konfig.Res_21 := FALSE;
   Zulauf_SF_Niv.Konfig.Res_22 := FALSE;
   Zulauf_SF_Niv.Konfig.Res_23 := FALSE;
   Zulauf_SF_Niv.Konfig.Res_24 := FALSE;
   Zulauf_SF_Niv.Konfig.Res_25 := FALSE;
   Zulauf_SF_Niv.Konfig.Res_26 := FALSE;
   Zulauf_SF_Niv.Konfig.Res_27 := FALSE;
   Zulauf_SF_Niv.Konfig.Res_28 := FALSE;
   Zulauf_SF_Niv.Konfig.Res_29 := FALSE;
   Zulauf_SF_Niv.Konfig.Res_30 := FALSE;
   Zulauf_SF_Niv.Konfig.Res_31 := FALSE;
   Zulauf_SF_Niv.MW_EW := 0.0;
   Zulauf_SF_Niv.MW_OG := 100.0;
   Zulauf_SF_Niv.MW_UG := 0.0;
   Zulauf_SF_Niv.GW_HH := 100.0;
   Zulauf_SF_Niv.GW_H := 100.0;
   Zulauf_SF_Niv.GW_L := 0.0;
   Zulauf_SF_Niv.GW_LL := 0.0;
   Zulauf_SF_Niv.GW_Hyst := 1.0;
   Zulauf_SF_Niv.VZ_St := 5;
   Zulauf_SF_Niv.VZ_Ex := 15;
   Zulauf_SF_Niv.MW_Avg := 30;
   Ablauf_NOx.Konfig.Peri := TRUE;
   Ablauf_NOx.Konfig.PW := FALSE;
   Ablauf_NOx.Konfig.Peri_0_20mA := FALSE;
   Ablauf_NOx.Konfig.Peri_4_20mA := TRUE;
   Ablauf_NOx.Konfig.Peri_PT100 := FALSE;
   Ablauf_NOx.Konfig.GW_Delta := FALSE;
   Ablauf_NOx.Konfig.Res_6 := FALSE;
   Ablauf_NOx.Konfig.Res_7 := FALSE;
   Ablauf_NOx.Konfig.Res_8 := FALSE;
   Ablauf_NOx.Konfig.Res_9 := FALSE;
   Ablauf_NOx.Konfig.Res_10 := FALSE;
   Ablauf_NOx.Konfig.Res_11 := FALSE;
   Ablauf_NOx.Konfig.Res_12 := FALSE;
   Ablauf_NOx.Konfig.Res_13 := FALSE;
   Ablauf_NOx.Konfig.Res_14 := FALSE;
   Ablauf_NOx.Konfig.Res_15 := FALSE;
   Ablauf_NOx.Konfig.Res_16 := FALSE;
   Ablauf_NOx.Konfig.Res_17 := FALSE;
   Ablauf_NOx.Konfig.Res_18 := FALSE;
   Ablauf_NOx.Konfig.Res_19 := FALSE;
   Ablauf_NOx.Konfig.Res_20 := FALSE;
   Ablauf_NOx.Konfig.Res_21 := FALSE;
   Ablauf_NOx.Konfig.Res_22 := FALSE;
   Ablauf_NOx.Konfig.Res_23 := FALSE;
   Ablauf_NOx.Konfig.Res_24 := FALSE;
   Ablauf_NOx.Konfig.Res_25 := FALSE;
   Ablauf_NOx.Konfig.Res_26 := FALSE;
   Ablauf_NOx.Konfig.Res_27 := FALSE;
   Ablauf_NOx.Konfig.Res_28 := FALSE;
   Ablauf_NOx.Konfig.Res_29 := FALSE;
   Ablauf_NOx.Konfig.Res_30 := FALSE;
   Ablauf_NOx.Konfig.Res_31 := FALSE;
   Ablauf_NOx.MW_EW := 0.0;
   Ablauf_NOx.MW_OG := 20.0;
   Ablauf_NOx.MW_UG := 0.0;
   Ablauf_NOx.GW_HH := 10.0;
   Ablauf_NOx.GW_H := 10.0;
   Ablauf_NOx.GW_L := 0.0;
   Ablauf_NOx.GW_LL := 0.0;
   Ablauf_NOx.GW_Hyst := 1.0;
   Ablauf_NOx.VZ_St := 5;
   Ablauf_NOx.VZ_Ex := 15;
   Ablauf_NOx.MW_Avg := 30;
   Ablauf_PO4.Konfig.Peri := TRUE;
   Ablauf_PO4.Konfig.PW := FALSE;
   Ablauf_PO4.Konfig.Peri_0_20mA := FALSE;
   Ablauf_PO4.Konfig.Peri_4_20mA := TRUE;
   Ablauf_PO4.Konfig.Peri_PT100 := FALSE;
   Ablauf_PO4.Konfig.GW_Delta := FALSE;
   Ablauf_PO4.Konfig.Res_6 := FALSE;
   Ablauf_PO4.Konfig.Res_7 := FALSE;
   Ablauf_PO4.Konfig.Res_8 := FALSE;
   Ablauf_PO4.Konfig.Res_9 := FALSE;
   Ablauf_PO4.Konfig.Res_10 := FALSE;
   Ablauf_PO4.Konfig.Res_11 := FALSE;
   Ablauf_PO4.Konfig.Res_12 := FALSE;
   Ablauf_PO4.Konfig.Res_13 := FALSE;
   Ablauf_PO4.Konfig.Res_14 := FALSE;
   Ablauf_PO4.Konfig.Res_15 := FALSE;
   Ablauf_PO4.Konfig.Res_16 := FALSE;
   Ablauf_PO4.Konfig.Res_17 := FALSE;
   Ablauf_PO4.Konfig.Res_18 := FALSE;
   Ablauf_PO4.Konfig.Res_19 := FALSE;
   Ablauf_PO4.Konfig.Res_20 := FALSE;
   Ablauf_PO4.Konfig.Res_21 := FALSE;
   Ablauf_PO4.Konfig.Res_22 := FALSE;
   Ablauf_PO4.Konfig.Res_23 := FALSE;
   Ablauf_PO4.Konfig.Res_24 := FALSE;
   Ablauf_PO4.Konfig.Res_25 := FALSE;
   Ablauf_PO4.Konfig.Res_26 := FALSE;
   Ablauf_PO4.Konfig.Res_27 := FALSE;
   Ablauf_PO4.Konfig.Res_28 := FALSE;
   Ablauf_PO4.Konfig.Res_29 := FALSE;
   Ablauf_PO4.Konfig.Res_30 := FALSE;
   Ablauf_PO4.Konfig.Res_31 := FALSE;
   Ablauf_PO4.MW_EW := 0.0;
   Ablauf_PO4.MW_OG := 20.0;
   Ablauf_PO4.MW_UG := 0.0;
   Ablauf_PO4.GW_HH := 15.0;
   Ablauf_PO4.GW_H := 15.0;
   Ablauf_PO4.GW_L := 0.0;
   Ablauf_PO4.GW_LL := 0.0;
   Ablauf_PO4.GW_Hyst := 1.0;
   Ablauf_PO4.VZ_St := 5;
   Ablauf_PO4.VZ_Ex := 15;
   Ablauf_PO4.MW_Avg := 30;
   Umwelt_WG.Konfig.Peri := TRUE;
   Umwelt_WG.Konfig.PW := FALSE;
   Umwelt_WG.Konfig.Peri_0_20mA := FALSE;
   Umwelt_WG.Konfig.Peri_4_20mA := TRUE;
   Umwelt_WG.Konfig.Peri_PT100 := FALSE;
   Umwelt_WG.Konfig.GW_Delta := FALSE;
   Umwelt_WG.Konfig.Res_6 := FALSE;
   Umwelt_WG.Konfig.Res_7 := FALSE;
   Umwelt_WG.Konfig.Res_8 := FALSE;
   Umwelt_WG.Konfig.Res_9 := FALSE;
   Umwelt_WG.Konfig.Res_10 := FALSE;
   Umwelt_WG.Konfig.Res_11 := FALSE;
   Umwelt_WG.Konfig.Res_12 := FALSE;
   Umwelt_WG.Konfig.Res_13 := FALSE;
   Umwelt_WG.Konfig.Res_14 := FALSE;
   Umwelt_WG.Konfig.Res_15 := FALSE;
   Umwelt_WG.Konfig.Res_16 := FALSE;
   Umwelt_WG.Konfig.Res_17 := FALSE;
   Umwelt_WG.Konfig.Res_18 := FALSE;
   Umwelt_WG.Konfig.Res_19 := FALSE;
   Umwelt_WG.Konfig.Res_20 := FALSE;
   Umwelt_WG.Konfig.Res_21 := FALSE;
   Umwelt_WG.Konfig.Res_22 := FALSE;
   Umwelt_WG.Konfig.Res_23 := FALSE;
   Umwelt_WG.Konfig.Res_24 := FALSE;
   Umwelt_WG.Konfig.Res_25 := FALSE;
   Umwelt_WG.Konfig.Res_26 := FALSE;
   Umwelt_WG.Konfig.Res_27 := FALSE;
   Umwelt_WG.Konfig.Res_28 := FALSE;
   Umwelt_WG.Konfig.Res_29 := FALSE;
   Umwelt_WG.Konfig.Res_30 := FALSE;
   Umwelt_WG.Konfig.Res_31 := FALSE;
   Umwelt_WG.MW_EW := 0.0;
   Umwelt_WG.MW_OG := 50.0;
   Umwelt_WG.MW_UG := 0.0;
   Umwelt_WG.GW_HH := 50.0;
   Umwelt_WG.GW_H := 50.0;
   Umwelt_WG.GW_L := 0.0;
   Umwelt_WG.GW_LL := 0.0;
   Umwelt_WG.GW_Hyst := 1.0;
   Umwelt_WG.VZ_St := 5;
   Umwelt_WG.VZ_Ex := 15;
   Umwelt_WG.MW_Avg := 30;
   Umwelt_WR.Konfig.Peri := TRUE;
   Umwelt_WR.Konfig.PW := FALSE;
   Umwelt_WR.Konfig.Peri_0_20mA := FALSE;
   Umwelt_WR.Konfig.Peri_4_20mA := TRUE;
   Umwelt_WR.Konfig.Peri_PT100 := FALSE;
   Umwelt_WR.Konfig.GW_Delta := FALSE;
   Umwelt_WR.Konfig.Res_6 := FALSE;
   Umwelt_WR.Konfig.Res_7 := FALSE;
   Umwelt_WR.Konfig.Res_8 := FALSE;
   Umwelt_WR.Konfig.Res_9 := FALSE;
   Umwelt_WR.Konfig.Res_10 := FALSE;
   Umwelt_WR.Konfig.Res_11 := FALSE;
   Umwelt_WR.Konfig.Res_12 := FALSE;
   Umwelt_WR.Konfig.Res_13 := FALSE;
   Umwelt_WR.Konfig.Res_14 := FALSE;
   Umwelt_WR.Konfig.Res_15 := FALSE;
   Umwelt_WR.Konfig.Res_16 := FALSE;
   Umwelt_WR.Konfig.Res_17 := FALSE;
   Umwelt_WR.Konfig.Res_18 := FALSE;
   Umwelt_WR.Konfig.Res_19 := FALSE;
   Umwelt_WR.Konfig.Res_20 := FALSE;
   Umwelt_WR.Konfig.Res_21 := FALSE;
   Umwelt_WR.Konfig.Res_22 := FALSE;
   Umwelt_WR.Konfig.Res_23 := FALSE;
   Umwelt_WR.Konfig.Res_24 := FALSE;
   Umwelt_WR.Konfig.Res_25 := FALSE;
   Umwelt_WR.Konfig.Res_26 := FALSE;
   Umwelt_WR.Konfig.Res_27 := FALSE;
   Umwelt_WR.Konfig.Res_28 := FALSE;
   Umwelt_WR.Konfig.Res_29 := FALSE;
   Umwelt_WR.Konfig.Res_30 := FALSE;
   Umwelt_WR.Konfig.Res_31 := FALSE;
   Umwelt_WR.MW_EW := 0.0;
   Umwelt_WR.MW_OG := 360.0;
   Umwelt_WR.MW_UG := 0.0;
   Umwelt_WR.GW_HH := 360.0;
   Umwelt_WR.GW_H := 360.0;
   Umwelt_WR.GW_L := 0.0;
   Umwelt_WR.GW_LL := 0.0;
   Umwelt_WR.GW_Hyst := 1.0;
   Umwelt_WR.VZ_St := 5;
   Umwelt_WR.VZ_Ex := 15;
   Umwelt_WR.MW_Avg := 5;
   Umwelt_LDr.Konfig.Peri := TRUE;
   Umwelt_LDr.Konfig.PW := FALSE;
   Umwelt_LDr.Konfig.Peri_0_20mA := FALSE;
   Umwelt_LDr.Konfig.Peri_4_20mA := TRUE;
   Umwelt_LDr.Konfig.Peri_PT100 := FALSE;
   Umwelt_LDr.Konfig.GW_Delta := FALSE;
   Umwelt_LDr.Konfig.Res_6 := FALSE;
   Umwelt_LDr.Konfig.Res_7 := FALSE;
   Umwelt_LDr.Konfig.Res_8 := FALSE;
   Umwelt_LDr.Konfig.Res_9 := FALSE;
   Umwelt_LDr.Konfig.Res_10 := FALSE;
   Umwelt_LDr.Konfig.Res_11 := FALSE;
   Umwelt_LDr.Konfig.Res_12 := FALSE;
   Umwelt_LDr.Konfig.Res_13 := FALSE;
   Umwelt_LDr.Konfig.Res_14 := FALSE;
   Umwelt_LDr.Konfig.Res_15 := FALSE;
   Umwelt_LDr.Konfig.Res_16 := FALSE;
   Umwelt_LDr.Konfig.Res_17 := FALSE;
   Umwelt_LDr.Konfig.Res_18 := FALSE;
   Umwelt_LDr.Konfig.Res_19 := FALSE;
   Umwelt_LDr.Konfig.Res_20 := FALSE;
   Umwelt_LDr.Konfig.Res_21 := FALSE;
   Umwelt_LDr.Konfig.Res_22 := FALSE;
   Umwelt_LDr.Konfig.Res_23 := FALSE;
   Umwelt_LDr.Konfig.Res_24 := FALSE;
   Umwelt_LDr.Konfig.Res_25 := FALSE;
   Umwelt_LDr.Konfig.Res_26 := FALSE;
   Umwelt_LDr.Konfig.Res_27 := FALSE;
   Umwelt_LDr.Konfig.Res_28 := FALSE;
   Umwelt_LDr.Konfig.Res_29 := FALSE;
   Umwelt_LDr.Konfig.Res_30 := FALSE;
   Umwelt_LDr.Konfig.Res_31 := FALSE;
   Umwelt_LDr.MW_EW := 0.0;
   Umwelt_LDr.MW_OG := 1100.0;
   Umwelt_LDr.MW_UG := 800.0;
   Umwelt_LDr.GW_HH := 1100.0;
   Umwelt_LDr.GW_H := 1100.0;
   Umwelt_LDr.GW_L := 800.0;
   Umwelt_LDr.GW_LL := 800.0;
   Umwelt_LDr.GW_Hyst := 1.0;
   Umwelt_LDr.VZ_St := 5;
   Umwelt_LDr.VZ_Ex := 15;
   Umwelt_LDr.MW_Avg := 30;
   Umwelt_LF.Konfig.Peri := TRUE;
   Umwelt_LF.Konfig.PW := FALSE;
   Umwelt_LF.Konfig.Peri_0_20mA := FALSE;
   Umwelt_LF.Konfig.Peri_4_20mA := TRUE;
   Umwelt_LF.Konfig.Peri_PT100 := FALSE;
   Umwelt_LF.Konfig.GW_Delta := FALSE;
   Umwelt_LF.Konfig.Res_6 := FALSE;
   Umwelt_LF.Konfig.Res_7 := FALSE;
   Umwelt_LF.Konfig.Res_8 := FALSE;
   Umwelt_LF.Konfig.Res_9 := FALSE;
   Umwelt_LF.Konfig.Res_10 := FALSE;
   Umwelt_LF.Konfig.Res_11 := FALSE;
   Umwelt_LF.Konfig.Res_12 := FALSE;
   Umwelt_LF.Konfig.Res_13 := FALSE;
   Umwelt_LF.Konfig.Res_14 := FALSE;
   Umwelt_LF.Konfig.Res_15 := FALSE;
   Umwelt_LF.Konfig.Res_16 := FALSE;
   Umwelt_LF.Konfig.Res_17 := FALSE;
   Umwelt_LF.Konfig.Res_18 := FALSE;
   Umwelt_LF.Konfig.Res_19 := FALSE;
   Umwelt_LF.Konfig.Res_20 := FALSE;
   Umwelt_LF.Konfig.Res_21 := FALSE;
   Umwelt_LF.Konfig.Res_22 := FALSE;
   Umwelt_LF.Konfig.Res_23 := FALSE;
   Umwelt_LF.Konfig.Res_24 := FALSE;
   Umwelt_LF.Konfig.Res_25 := FALSE;
   Umwelt_LF.Konfig.Res_26 := FALSE;
   Umwelt_LF.Konfig.Res_27 := FALSE;
   Umwelt_LF.Konfig.Res_28 := FALSE;
   Umwelt_LF.Konfig.Res_29 := FALSE;
   Umwelt_LF.Konfig.Res_30 := FALSE;
   Umwelt_LF.Konfig.Res_31 := FALSE;
   Umwelt_LF.MW_EW := 0.0;
   Umwelt_LF.MW_OG := 100.0;
   Umwelt_LF.MW_UG := 0.0;
   Umwelt_LF.GW_HH := 100.0;
   Umwelt_LF.GW_H := 100.0;
   Umwelt_LF.GW_L := 0.0;
   Umwelt_LF.GW_LL := 0.0;
   Umwelt_LF.GW_Hyst := 1.0;
   Umwelt_LF.VZ_St := 5;
   Umwelt_LF.VZ_Ex := 15;
   Umwelt_LF.MW_Avg := 30;
   Umwelt_T.Konfig.Peri := TRUE;
   Umwelt_T.Konfig.PW := FALSE;
   Umwelt_T.Konfig.Peri_0_20mA := FALSE;
   Umwelt_T.Konfig.Peri_4_20mA := TRUE;
   Umwelt_T.Konfig.Peri_PT100 := FALSE;
   Umwelt_T.Konfig.GW_Delta := FALSE;
   Umwelt_T.Konfig.Res_6 := FALSE;
   Umwelt_T.Konfig.Res_7 := FALSE;
   Umwelt_T.Konfig.Res_8 := FALSE;
   Umwelt_T.Konfig.Res_9 := FALSE;
   Umwelt_T.Konfig.Res_10 := FALSE;
   Umwelt_T.Konfig.Res_11 := FALSE;
   Umwelt_T.Konfig.Res_12 := FALSE;
   Umwelt_T.Konfig.Res_13 := FALSE;
   Umwelt_T.Konfig.Res_14 := FALSE;
   Umwelt_T.Konfig.Res_15 := FALSE;
   Umwelt_T.Konfig.Res_16 := FALSE;
   Umwelt_T.Konfig.Res_17 := FALSE;
   Umwelt_T.Konfig.Res_18 := FALSE;
   Umwelt_T.Konfig.Res_19 := FALSE;
   Umwelt_T.Konfig.Res_20 := FALSE;
   Umwelt_T.Konfig.Res_21 := FALSE;
   Umwelt_T.Konfig.Res_22 := FALSE;
   Umwelt_T.Konfig.Res_23 := FALSE;
   Umwelt_T.Konfig.Res_24 := FALSE;
   Umwelt_T.Konfig.Res_25 := FALSE;
   Umwelt_T.Konfig.Res_26 := FALSE;
   Umwelt_T.Konfig.Res_27 := FALSE;
   Umwelt_T.Konfig.Res_28 := FALSE;
   Umwelt_T.Konfig.Res_29 := FALSE;
   Umwelt_T.Konfig.Res_30 := FALSE;
   Umwelt_T.Konfig.Res_31 := FALSE;
   Umwelt_T.MW_EW := 0.0;
   Umwelt_T.MW_OG := 70.0;
   Umwelt_T.MW_UG := -30.0;
   Umwelt_T.GW_HH := 40.0;
   Umwelt_T.GW_H := 35.0;
   Umwelt_T.GW_L := -2.0;
   Umwelt_T.GW_LL := -10.0;
   Umwelt_T.GW_Hyst := 1.0;
   Umwelt_T.VZ_St := 5;
   Umwelt_T.VZ_Ex := 15;
   Umwelt_T.MW_Avg := 30;
   Ablauf_LF.Konfig.Peri := TRUE;
   Ablauf_LF.Konfig.PW := FALSE;
   Ablauf_LF.Konfig.Peri_0_20mA := FALSE;
   Ablauf_LF.Konfig.Peri_4_20mA := TRUE;
   Ablauf_LF.Konfig.Peri_PT100 := FALSE;
   Ablauf_LF.Konfig.GW_Delta := FALSE;
   Ablauf_LF.Konfig.Res_6 := FALSE;
   Ablauf_LF.Konfig.Res_7 := FALSE;
   Ablauf_LF.Konfig.Res_8 := FALSE;
   Ablauf_LF.Konfig.Res_9 := FALSE;
   Ablauf_LF.Konfig.Res_10 := FALSE;
   Ablauf_LF.Konfig.Res_11 := FALSE;
   Ablauf_LF.Konfig.Res_12 := FALSE;
   Ablauf_LF.Konfig.Res_13 := FALSE;
   Ablauf_LF.Konfig.Res_14 := FALSE;
   Ablauf_LF.Konfig.Res_15 := FALSE;
   Ablauf_LF.Konfig.Res_16 := FALSE;
   Ablauf_LF.Konfig.Res_17 := FALSE;
   Ablauf_LF.Konfig.Res_18 := FALSE;
   Ablauf_LF.Konfig.Res_19 := FALSE;
   Ablauf_LF.Konfig.Res_20 := FALSE;
   Ablauf_LF.Konfig.Res_21 := FALSE;
   Ablauf_LF.Konfig.Res_22 := FALSE;
   Ablauf_LF.Konfig.Res_23 := FALSE;
   Ablauf_LF.Konfig.Res_24 := FALSE;
   Ablauf_LF.Konfig.Res_25 := FALSE;
   Ablauf_LF.Konfig.Res_26 := FALSE;
   Ablauf_LF.Konfig.Res_27 := FALSE;
   Ablauf_LF.Konfig.Res_28 := FALSE;
   Ablauf_LF.Konfig.Res_29 := FALSE;
   Ablauf_LF.Konfig.Res_30 := FALSE;
   Ablauf_LF.Konfig.Res_31 := FALSE;
   Ablauf_LF.MW_EW := 0.0;
   Ablauf_LF.MW_OG := 2000.0;
   Ablauf_LF.MW_UG := 0.0;
   Ablauf_LF.GW_HH := 2000.0;
   Ablauf_LF.GW_H := 2000.0;
   Ablauf_LF.GW_L := 0.0;
   Ablauf_LF.GW_LL := 0.0;
   Ablauf_LF.GW_Hyst := 1.0;
   Ablauf_LF.VZ_St := 5;
   Ablauf_LF.VZ_Ex := 15;
   Ablauf_LF.MW_Avg := 15;

END_DATA_BLOCK

DATA_BLOCK "DB117_MW_EA"
{ S7_Optimized_Access := 'FALSE' }
VERSION : 0.1
NON_RETAIN
   STRUCT
      Zulauf_AR_Niv : "T_MW_EA";   // Zulauf - Pumpwerk "Alter Rechen" - Niveau
      Zulauf_AR_Temp : "T_MW_EA";   // Zulauf - Pumpwerk "Alter Rechen" - Temperatur
      Zulauf_AR_DF : "T_MW_EA";   // Zulauf - Pumpwerk "Alter Rechen" - Durchfluss
      BB1_AS1_SS : "T_MW_EA";   // Becken 1 - Ablaufschieber 1 - Schieberstellung
      BB1_AS2_SS : "T_MW_EA";   // Becken 1 - Ablaufschieber 2 - Schieberstellung
      BB2_AS1_SS : "T_MW_EA";   // Becken 2 - Ablaufschieber 1 - Schieberstellung
      BB2_AS2_SS : "T_MW_EA";   // Becken 2 - Ablaufschieber 2 - Schieberstellung
      BB1_O2 : "T_MW_EA";   // Becken 1 - O2-Gehalt
      BB1_Temp : "T_MW_EA";   // Becken 1 - Temperatur
      BB2_O2 : "T_MW_EA";   // Becken 2 - O2-Gehalt
      BB2_Temp : "T_MW_EA";   // Becken 2 - Temperatur
      BB1_DF : "T_MW_EA";   // Becken 1 - Ablauf - Durchfluss
      BB2_DF : "T_MW_EA";   // Becken 2 - Ablauf - Durchfluss
      Zulauf_Niv : "T_MW_EA";   // Zulauf - Vorlagebehälter - Niveau
      Zulauf_DF : "T_MW_EA";   // Zulauf - Rechen - Durchfluss
      Verteiler_pH : "T_MW_EA";   // Zulauf - Verteiler - pH-Wert
      Verteiler_O2 : "T_MW_EA";   // Zulauf - Verteiler  - O2-Gehalt
      Verteiler_Temp : "T_MW_EA";   // Zulauf - Verteiler - Temperatur
      BB_UeSS_DF : "T_MW_EA";   // Becken 1+2 - Ablauf ÜSS - Durchfluss
      Ablauf_DF : "T_MW_EA";   // Ablauf - Durchfluss
      Ablauf_pH : "T_MW_EA";   // Ablauf - pH-Wert
      Ablauf_O2 : "T_MW_EA";   // Ablauf - O2-Gehalt
      Ablauf_Temp : "T_MW_EA";   // Ablauf - Temperatur
      Schlamm_ED_Niv : "T_MW_EA";   // Schlamm - Eindicker - Niveau
      Schlamm_Besch_Niv : "T_MW_EA";   // Schlamm - Beschickung - Niveau
      Schlamm_Besch_DF : "T_MW_EA";   // Schlamm - Beschickung - Durchfluss
      Truebwasser_Niv : "T_MW_EA";   // Trübwasserpumpwerk - Niveau
      Truebwasser_DF : "T_MW_EA";   // Trübwasserpumpwerk - Durchfluss
      Zulauf_SF_Niv : "T_MW_EA";   // Zulauf - Sandfang - Niveau
      Ablauf_NOx : "T_MW_EA";   // Ablauf - Dortmundbrunnen - Nitratmessung
      Ablauf_PO4 : "T_MW_EA";   // Ablauf - Dortmundbrunnen - Phosphatmessung
      Umwelt_WG : "T_MW_EA";   // Wetterstation - Windgeschwindigkeit
      Umwelt_WR : "T_MW_EA";   // Wetterstation - Windrichtung
      Umwelt_LDr : "T_MW_EA";   // Wetterstation - Luftdruck
      Umwelt_LF : "T_MW_EA";   // Wetterstation - Luftfeuchtigkeit
      Umwelt_T : "T_MW_EA";   // Wetterstation - Temperatur
      Ablauf_LF : "T_MW_EA";   // Ablauf - Leitfähigkeit
   END_STRUCT;


